DATA_BLOCK "DOOR_CLEANER_MOTOR_DB"	// DB 10
AUTHOR : Kamillas
VERSION : 0.1
  STRUCT
   DC_MTR_RDY_FOR_STA : BOOL ;	//DOOR CLEANER READY FOR START
   DC_MTR_UP_RUN_FB : BOOL ;	//DOOR CLEANER UP RUNNING FEED BACK
   DC_MTR_OLR_TRIP : BOOL ;	//DOOR CLEANER OVER LOAD TRIP
   DC_MTR_DN_RUN_FB : BOOL ;	//DOOR CLEANER DOWN RUNNING FEED BACK
   DC_MTR_AUTO_SS : BOOL ;	//DOOR CLEANER AUTO SELECTOR SWITCH
   DC_MTR_MAN_SS : BOOL ;	//DOOR CLEANER MANUAL SELECTOR SWITCH
   DC_MTR_UP_STA_PB : BOOL ;	//DOOR CLEANER UP START PUSH BUTTON
   DC_MTR_DN_STA_PB : BOOL ;	//DOOR CLEANER DOWN START PUSH BUTTON
   DC_MTR_STP_PB : BOOL ;	//DOOR CLEANER STOP PUSH BUTTON
   DC_MTR_HME_PB : BOOL ;	//DOOR CLEANER HOME PUSH BUTTON
   DC_MTR_UP_LS : BOOL ;	//DOOR CLEANER UP LIMIT SWITCH
   DC_MTR_DN_LS : BOOL ;	//DOOR CLEANER DOWN LIMIT SWITCH
   DC_MTR_HME_LS : BOOL ;	//DOOR CLEANER HOME LIMIT SWITCH
   CLN_OVN_DR_STA_PB : BOOL ;	//CLEAN OVEN DOOR START PUSH BUTTON
   CLN_OVN_DR_STP_PB : BOOL ;	//CLEAN OVEN DOOR STOP PUSH BUTTON
   DC_MTR_UP_ON_CMD : BOOL ;	//DOOR CLEANER UP ON COMMAND
   DC_MTR_DN_ON_CMD : BOOL ;	//DOOR CLEANER DOWN ON COMMAND
   DC_MTR_UP_IND : BOOL ;	//DOOR CLEANER UP INDICATOR
   DC_MTR_DN_IND : BOOL ;	//DOOR CLEANER DOWN INDICATOR
   DC_MTR_HME_IND : BOOL ;	//DOOR CLEANER HOME INDICATOR
   CLN_OVN_DR_AUTO_IND : BOOL ;	//CLEAN OVEN DOOR AUTO INDICATOR
   DC_MTR_FLT : BOOL ;	//DOOR COMPRESSOR MOTOR FAULT
   DC_MTR_FLT_TMR : INT ;	//DOOR COMPRESSOR MOTOR FAULT TIMER
   DC_MTR_FLT_GEN_TIME : INT  := 3;	//DOOR COMPRESSOR MOTOR FAULT GEMERATION TIME
   PULSE_1 : BOOL ;	//PULSE 1
   PULSE_2 : BOOL ;	//PULSE 2
   PULSE_3 : BOOL ;	//PULSE 3
   PULSE_4 : BOOL ;	//PULSE 4
   PULSE_5 : BOOL ;	//PULSE 5
   PULSE_6 : BOOL ;	//PULSE 6
   PULSE_7 : BOOL ;	//PULSE 7
   PULSE_8 : BOOL ;	//PULSE 8
   DC_MTR_ILK_BIT : BOOL ;	//DOOR CLEANER MOTOR INTERLOCK BIT
   DC_MTR_AUTO_STA_BIT : BOOL ;	//DOOR CLEANER MOTOR AUTO START BIT
   DC_MTR_HME_POS_BIT : BOOL ;	//DOOR CLEANER MOTOR HOME POSITION BIT
   DC_MTR_UP_DN_CNT_OVR : BOOL ;	//DOOR CLEANER MOTOR UP DOWN COUNT OVER
   DC_MTR_UP_DN_CNT : INT ;	//DOOR CLEANER UP DOWN COUNT
   DC_MTR_UP_DN_CNT_SET : INT  := 2;	//DOOR CLEANER MOTOR UP DOWN COUNT SET POINT
   DC_MTR_LOC_SS : BOOL ;	//DOOR CLEANER MOTOR LOCAL SELECTOR SWITCH
   DC_MTR_HME_ON_CMD : BOOL ;	//DOOR CLEANER HOME ON COMMAND
   DC_MTR_CLN_OVN_DOOR_IND : BOOL ;	//DOOR CLEANER - CLEAN OVEN DOOR INDICATOR
   TRA_SLOW_FWD_OP_CUT : BOOL ;	//TRAVEL SLOW FORWARD OUTPUT CUT
   TRA_SLOW_FWD_FLT_TMR : INT ;	//TRAVEL SLOW FORWARD FAULT TIMER
   TRA_SLOW_FWD_FLT_GEN : INT  := 8;	//TRAVEL SLOW FORWARD FAULT GENERATION TIME
   TRA_SLOW_FWD_OP_CT_TM : INT ;	//TRAVEL SLOW FORWARD OUTPUT CUT TIMER
   TRA_SLOW_FWD_FLT : BOOL ;	//TRAVEL SLOW FORWARD FAULT
   TRA_SLOW_AUTO_FWD_OVR : BOOL ;	//TRAVEL SLOW AUTO FORWARD OVER
   TRA_SLOW_AUTO_FWD_DEL : INT  := 3;	//TRAVEL SLOW AUTO FORWARD OVER DELAY
   TRA_SLOW_ATO_FWD_DL_T : INT ;	//TRAVEL SLOW AUTO FORWARD OVER DELAY TIMER
   TRA_SLOW_RET_OP_CUT : BOOL ;	//TRAVEL SLOW RETRACT OUTPUT CUT
   TRA_SLOW_RET_FLT_TMR : INT ;	//TRAVEL SLOW RETRACT FAULT TIMER
   TRA_SLOW_RET_FLT_GEN : INT  := 8;	//TRAVEL SLOW RETRACT FAULT GENERATION TIME
   TRA_SLOW_RET_OP_CT_TM : INT ;	//TRAVEL SLOW RETRACT OUTPUT CUT TIMER
   TRA_SLOW_RET_FLT : BOOL ;	//TRAVEL SLOW RETRACT FAULT
   TRA_SLOW_AUTO_RET_OVR : BOOL ;	//TRAVEL SLOW AUTO RETRACT OVER
   TRA_SLOW_AUTO_RET_DEL : INT  := 3;	//TRAVEL SLOW AUTO RETRACT OVER DELAY
   TRA_SLOW_ATO_RET_DL_T : INT ;	//TRAVEL SLOW AUTO RETRACT OVER DELAY TIMER
   TRA_NOR_FWD_OP_CUT : BOOL ;	//TRAVEL NORMAL FORWARD OUTPUT CUT
   TRA_NOR_FWD_FLT_TMR : INT ;	//TRAVEL NORMAL FORWARD FAULT TIMER
   TRA_NOR_FWD_FLT_GEN : INT  := 8;	//TRAVEL NORMAL FORWARD FAULT GENERATION TIME
   TRA_NOR_FWD_OP_CT_TM : INT ;	//TRAVEL NORMAL FORWARD OUTPUT CUT TIMER
   TRA_NOR_FWD_FLT : BOOL ;	//TRAVEL NORMAL FORWARD FAULT
   TRA_NOR_AUTO_FWD_OVR : BOOL ;	//TRAVEL NORMAL AUTO FORWARD OVER
   TRA_NOR_AUTO_FWD_DEL : INT  := 3;	//TRAVEL NORMAL AUTO FORWARD OVER DELAY
   TRA_NOR_ATO_FWD_DL_T : INT ;	//TRAVEL NORMAL AUTO FORWARD OVER DELAY TIMER
   TRA_NOR_RET_OP_CUT : BOOL ;	//TRAVEL NORMAL RETRACT OUTPUT CUT
   TRA_NOR_RET_FLT_TMR : INT ;	//TRAVEL NORMAL RETRACT FAULT TIMER
   TRA_NOR_RET_FLT_GEN : INT  := 8;	//TRAVEL NORMAL RETRACT FAULT GENERATION TIME
   TRA_NOR_RET_OP_CT_TM : INT ;	//TRAVEL NORMAL RETRACT OUTPUT CUT TIMER
   TRA_NOR_RET_FLT : BOOL ;	//TRAVEL NORMAL RETRACT FAULT
   TRA_NOR_AUTO_RET_OVR : BOOL ;	//TRAVEL NORMAL AUTO RETRACT OVER
   TRA_NOR_AUTO_RET_DEL : INT  := 3;	//TRAVEL NORMAL AUTO RETRACT OVER DELAY
   TRA_NOR_ATO_RET_DL_T : INT ;	//TRAVEL NORMAL AUTO RETRACT OVER DELAY TIMER
   TRA_SLOW_FWD_CMD : BOOL ;	//TRAVEL SLOW FORWARD COMMAND
   TRA_SLOW_RET_CMD : BOOL ;	//TRAVEL SLOW RETRACT COMMAND
   TRA_NOR_FWD_CMD : BOOL ;	//TRAVEL NORMAL FORWARD COMMAND
   TRA_NOR_RET_CMD : BOOL ;	//TRAVEL NORMAL RETRACT COMMAND
   TRA_RELIVE_CMD : BOOL ;	//TRAVEL RELIVE COOMMAND
   TRA_AUTO_FWD_CLN_POS_SET : BOOL ;	//TRAVEL AUTO FORWARD TO CLEANING POSITION SET
   TRA_AUTO_RET_SET : BOOL ;	//TRAVEL AUTO RETRACT SET
   TRA_CLN_POS_LS : BOOL ;	//TRAVEL CLEANING POSTION LIMIT SWITCH
   PULSE_9 : BOOL ;	//PULSE 9
   PULSE_10 : BOOL ;	//PULSE 10
   PULSE_11 : BOOL ;	//PULSE 11
   PULSE_12 : BOOL ;	//PULSE 12
   PULSE_13 : BOOL ;	//PULSE 13
   PULSE_14 : BOOL ;	//PULSE 14
   PULSE_15 : BOOL ;	//PULSE 15
   PULSE_16 : BOOL ;	//PULSE 16
   DC_MTR_HME_SET : BOOL ;	//TRAVEL AUTO HOME SET
   DC_MTR_AUTO_OPER_FIN : BOOL ;	//DOOR CLEANER MOTOR AUTO OPERATIONS FINISHED
   DC_AUTO_STOPPED : BOOL ;	//DOOR CLEANER OPERATIONS STOPED WHILE IN AUTO OPERATION
   DC_MTR_UP_LS_HOLD : BOOL ;	//UP LIMIT SWITCH HOLDING
   DC_MTR_DN_LS_HOLD : BOOL ;	//DOWN LIMIT SWITCH HOLDING
   DC_MTR_HME_LS_HOLD : BOOL ;	//HOME LIMIT SWITCH HOLDING
  END_STRUCT ;	
BEGIN
   DC_MTR_FLT_GEN_TIME := 3;
   DC_MTR_UP_DN_CNT_SET := 2;
   TRA_SLOW_FWD_FLT_GEN := 8;
   TRA_SLOW_AUTO_FWD_DEL := 3;
   TRA_SLOW_RET_FLT_GEN := 8;
   TRA_SLOW_AUTO_RET_DEL := 3;
   TRA_NOR_FWD_FLT_GEN := 8;
   TRA_NOR_AUTO_FWD_DEL := 3;
   TRA_NOR_RET_FLT_GEN := 8;
   TRA_NOR_AUTO_RET_DEL := 3;
END_DATA_BLOCK

DATA_BLOCK "WIN_CC_DB"	// DB 11
AUTHOR : Kamilas
VERSION : 0.1
  STRUCT
   MAIN_PWR_ON_PB : BOOL ;	//MAIN POWER ON PUSH BUTTON
   MAIN_PWR_OFF_PB : BOOL ;	//MAIN POWER OFF PUSH BUTTON
   MP_LAMP_TEST_PB : BOOL ;	//MAIN POWER LAMP TEST PUSH BUTTON
   MP_ALARM_ACK_PB : BOOL ;	//MAIN POWER ALARM ACKNOWLEDGE PUSH BUTTON
   CTRL_SELECTION_CD : BOOL ;	//CONTROL SELECTRION CD
   ALL_MECH_QUICK_STP : BOOL ;	//ALL MECHANICAL QUICK STOP
   REP_MAN_SS : BOOL ;	//REPAIR MANUAL SELECTION
   SEMI_AUTO_SS : BOOL ;	//SEMI AUTO SELECTION
   PUMP_1_RDY_FOR_STA : BOOL ;	//PUMP 1 READY FOR START
   PUMP_2_RDY_FOR_STA : BOOL ;	//PUMP 2 READY FOR START
   CIR_PUMP_RDY_FOR_STA : BOOL ;	//CIRCULATION PUMP READY FOR START
   COLR_FAN_RDY_FOR_STA : BOOL ;	//COOLER FAN READY FOR START
   CD_LCS_SS : BOOL ;	//CONTROL DESK / LOCAL CONTROL SELECTOR SWITCH
   HY_PUMP_1_2_SS : BOOL ;	//PUMP 1 OR 2 SELECTOR SWITCH
   HY_PUMP_1_STA_PB : BOOL ;	//PUMP 1 START PUSH BUTTON
   HY_PUMP_1_STP_PB : BOOL ;	//PUMP 1 STOP PUSH BUTTON
   HY_PUMP_2_STA_PB : BOOL ;	//PUMP 2 START PUSH BUTTON
   HY_PUMP_2_STP_PB : BOOL ;	//PUMP 2 STOP PUSH BUTTON
   HY_PUMP_1_2_SS_LCS : BOOL ;	//PUMP 1 OR 2 SELECTOR SWITCH LCS
   HY_PUMP_1_STA_PB_LCS : BOOL ;	//PUMP 1 START PUSH BUTTON LCS
   HY_PUMP_1_STP_PB_LCS : BOOL ;	//PUMP 1 STOP PUSH BUTTON LCS
   HY_PUMP_2_STA_PB_LCS : BOOL ;	//PUMP 2 START PUSH BUTTON LCS
   HY_PUMP_2_STP_PB_LCS : BOOL ;	//PUMP 2 STOP PUSH BUTTON LCS
   HY_CIR_PUMP_STA_PB_LCS : BOOL ;	//CIRCULATION PUMP START PUSH BUTTON LCS
   HY_CIR_PUMP_STP_PB_LCS : BOOL ;	//CIRCULATION PUMP STOP PUSH BUTTON LCS
   HY_COLR_FAN_STA_PB_LCS : BOOL ;	//COOLER FAN START PUSH BUTTON LCS
   HY_COLR_FAN_STP_PB_LCS : BOOL ;	//COOLER FAN STOP PUSH BUTTON LCS
   TRA_DRV_1_BRK_RDY_FOR_ST : BOOL ;	//TRAVEL GROUP 1 BREAK READY FOR START
   TRA_DRV_2_BRK_RDY_FOR_ST : BOOL ;	//TRAVEL GROUP 2 BREAK READY FOR START
   TRA_MODE_AUTO_MAN_SS : BOOL ;	//TRAVEL MODE AUTO/MANUAL BUTTON
   TRA_DRV_1_PROF_HARD_SS : BOOL ;	//TRAVEL DRIVE 1 PROFIBUS/HARD WIRE SELECTRO SWITCH
   TRA_DRV_1_RDY_FOR_STA : BOOL ;	//TRAVEL DRIVE 1 READY FOR START
   TRA_DRV_2_PROF_HARD_SS : BOOL ;	//TRAVEL DRIVE 2 PROFIBUS/HARD WIRE SELECTRO SWITCH
   TRA_DRV_2_RDY_FOR_STA : BOOL ;	//TRAVEL DRIVE 2 READY FOR START
   AC_MTR_RDY_FOR_STA : BOOL ;	//AIR COMPRESSOR MOTOR READY FOR START
   AC_MTR_STA_PB : BOOL ;	//AIR COMPRESSOR MOTOR START PUSH BUTTON
   AC_MTR_STP_PB : BOOL ;	//AIR COMPRESSOR MOTOR STOP PUSH BUTTON
   IDF_DRV_RDY_FOR_STA : BOOL ;	//ID FAN DRIVE READY FOR START
   WTR_PMP_MTR_RDY_FOR_STA : BOOL ;	//WATER PUMP MOTOR READY FOR START
   HOOD_STA_PB : BOOL ;	//HOOD START PUSH BUTTON
   HOOD_STP_PB : BOOL ;	//HOOD STOP PUSH BUTTON
   IDF_DRV_LS_HS_SEL : BOOL ;	//ID FAN DRIVE LOW SPEED/HIGH SPEED SELECTION
   DE_DOOR_EXT_LOC_SS : BOOL ;	//DOOR EXTRACTOR LOCAL SELECTOR SWITCH
   DE_DOOR_EXT_MAN_SS : BOOL ;	//DOOR EXTRACTOR MANUAL SELECTOR SWITCH
   DE_DOOR_EXT_AUTO_SS : BOOL ;	//DOOR EXTRACTOR AUTO SELECTOR SWITCH
   DE_DOOR_EXT_STP_PB : BOOL ;	//DOOR EXTRACTOR STOP PUSH BUTTON
   DE_SLEW_FWD_STA_PB : BOOL ;	//SLEW FORWARD START PUSH BUTTON
   DE_SLEW_RET_STA_PB : BOOL ;	//SLEW RETRACT START
   DE_VER_COMP_FWD_STA_PB : BOOL ;	//VERTICAL COMPENSATION FORWARD START PUSH BUTTON
   DE_VER_COMP_RET_STA_PB : BOOL ;	//VERTICAL COMPENSATION RETRACT START PUSH BUTTON
   DE_TRA_FWD_STA_PB : BOOL ;	//TRAVEL FORWARD START PUSH BUTTON
   DE_TRA_RET_STA_PB : BOOL ;	//TRAVEL RETRACT START PUSH BUTTON
   MAIN_STK_UP_STA_PB : BOOL ;	//MAIN STROKE UP START PUSH BUTTON
   MAIN_STK_DN_PB : BOOL ;	//MAIN STROKE DOWN START PUSH BUTTON
   FIN_STK_UP_STA_PB : BOOL ;	//FINAL STROKE UP START PUSH BUTTON
   FIN_STK_DN_PB : BOOL ;	//FINAL STROKE DOWN START PUSH BUTTON
   PRE_STK_UP_STA_PB : BOOL ;	//PRE STROKE UP START PUSH BUTTON
   PRE_STK_UP_DN_PB : BOOL ;	//PRE STROKE DOWN START PUSH BUTTON
   DR_SPNG_LK_STA_PB : BOOL ;	//DOOR SPRING PRESSURE START PUSH BUTTON
   DR_SPNG_UNLK_STA_PB : BOOL ;	//DOOR SPRING PRESSURE RELEASE START PUSH BUTTON
   DR_LCH_TURN_UP_PB : BOOL ;	//DOOR LATCH TURNING LOCK PUSH BUTTON
   DR_LCH_TURN_DN_PB : BOOL ;	//DOOR LATCH TURNING UNLOCK PUSH BUTTON
   JC_CRA_TRA_FWD_STA_PB : BOOL ;	//JAMB CLEANER CARRIAGE TRAVEL FORWARD PUSH BUTTON
   JC_CRA_TRA_RET_STA_PB : BOOL ;	//JAMB CLEANER CARRIAGE TRAVEL RETRACT PUSH BUTTON
   JC_VC_UP_STA_PB : BOOL ;	//JAMB CLEANER VERTICAL CLEANER UP START PUSH BUTTON
   JC_VC_DN_STA_PB : BOOL ;	//JAMB CLEANER VERTICAL CLEANER DOWN START PUSH BUTTON
   JC_STP_PB : BOOL ;	//JAMB CLEANER OPERATIONS STOP PUSH BUTTON
   JC_VC_HME_STA_PB : BOOL ;	//JAMB CLEANER VERTICAL CLEANER HOME START PUSH BUTTON
   CLN_OVN_JMB_STA_PB : BOOL ;	//CLEAN OVEN JAMB AUTO START PUSH BUTTON
   CLN_OVN_JMB_STP_PB : BOOL ;	//CLEAN OVEN JAMB AUTO STOP PUSH BUTTON
   JC_AUTO_SS : BOOL ;	//JAMB CLEANER AUTO MODE SELECTOR SWITCH
   JC_MAN_SS : BOOL ;	//JAMB CLEANER MANUAL MODE SELECTOR SWITCH
   JC_LOC_SS : BOOL ;	//JAMB CLEANER LOCAL MODE SELECTOR SWITCH
   JC_AUTO_STA_PB : BOOL ;	//JAMB CLEANER AUTO START PUSH BUTTON
   GC_AUTO_SS : BOOL ;	//GUIDE CAGE AUTO SELECTOR SWITCH
   GC_MAN_SS : BOOL ;	//GUIDE CAGE MANUAL SELECTOR SWITCH
   GC_TRA_FWD_STA_PB : BOOL ;	//GUIDE CAGE TRAVEL FORWARD START PUSH BUTTON
   GC_TRA_RET_STA_PB : BOOL ;	//GUIDE CAGE TRAVEL RETRACT START PUSH BUTTON
   GC_STP_PB : BOOL ;	//GUIDE CAGE AUTO STOP PUSH BUTTON
   GC_TRA_AUTO_STA_PB : BOOL ;	//GUIDE CAGE TRAVEL AUTO START PUSH BUTTON
   GC_TRA_AUTO_STP_PB : BOOL ;	//GUIDE CAGE TRAVEL AUTO STOP PUSH BUTTON
   GC_AUTO_STA_PB : BOOL ;	//GUIDE CAGE AUTO START PUSH BUTTON
   DC_MTR_RDY_FOR_STA : BOOL ;	//DOOR CLEANER READY FOR START
   DC_MTR_AUTO_SS : BOOL ;	//DOOR CLEANER AUTO SELECTOR SWITCH
   DC_MTR_MAN_SS : BOOL ;	//DOOR CLEANER MANUAL SELECTOR SWITCH
   DC_MTR_UP_STA_PB : BOOL ;	//DOOR CLEANER UP START PUSH BUTTON
   DC_MTR_DN_STA_PB : BOOL ;	//DOOR CLEANER DOWN START PUSH BUTTON
   DC_MTR_STP_PB : BOOL ;	//DOOR CLEANER STOP PUSH BUTTON
   DC_MTR_HME_PB : BOOL ;	//DOOR CLEANER HOME PUSH BUTTON
   CLN_OVN_DR_STA_PB : BOOL ;	//CLEAN OVEN DOOR START PUSH BUTTON
   CLN_OVN_DR_STP_PB : BOOL ;	//CLEAN OVEN DOOR STOP PUSH BUTTON
   DC_MTR_LOC_SS : BOOL ;	//DOOR CLEANER MOTOR LOCAL SELECTOR SWITCH
   SP_STP_PB : BOOL ;	//SERVICE PLATFORM STOP PUSH BUTTON
   SP_STA_PB : BOOL ;	//SERVICE PLATFORM START PUSH BUTTON
   EMG_ACCM_STA_PB_LCS : BOOL ;	//EMERGENCY ACCUMULATOR START PUSH BUTTON LCS
   EMG_ACCM_STP_PB_LCS : BOOL ;	//EMERGENCY ACCUMULATOR STOP PUSH BUTTON LCS
   EXT_OVN_DOR_STA_PB : BOOL ;	//EXTRACT OVEN DOOR START PUSH BUTTON
   EXT_RPL_FUNC_STP_PB : BOOL ;	//EXTRACT AND REPLACE FUNCTIONAL STOP PUSH BUTTON
   RPL_OVN_DOR_STA_PB : BOOL ;	//REPLACE OVEN DOOR START PUSH BUTTON
   ALL_OPER_IN_OPER_MODE : BOOL ;	//ALL OPERATION IN OPERATION MODE
   ALL_OPER_IN_REP_MODE : BOOL ;	//ALL OPERATION IN REPAIR MODE
   SP_TRA_FWD_STA_PB : BOOL ;	//SERVICE PLATFORM TRAVEL FORWARD START PUSH BUTTON
   SP_TRA_REV_STA_PB : BOOL ;	//SERVICE PLATFORM TRAVEL REVERSE START PUSH BUTTON
   EMERGENCY_STOP : BOOL ;	//EMERGENCY STOP
   HY_LAMP_TEST : BOOL ;	//HYDRALIC SYSTEM LAMP PUSH BUTTON
   SP_AUTO_STP_PB : BOOL ;	//SERVICE PLATFORM AUTO STOP PUSH BUTTON
   SP_TRA_AUTO_STA_PB : BOOL ;	//SERVICE PLATFORM TRAVEL AUTO START PUSH BUTTON
   SP_TRA_AUTO_STP_PB : BOOL ;	//SERVICE PLATFORM TRAVEL AUTO STOP PUSH BUTTON
   SP_AUTO_STA_PB : BOOL ;	//SERVICE PLATFORM AUTO START PUSH BUTTON
   SP_AUTO_SS : BOOL ;	//SERVICE PLATFORM AUTO MODE SELECTOR SWITCH
   SP_MAN_SS : BOOL ;	//SERVICE PLATFORM MANUAL MODE SELECTOR SWITCH
   MAIN_PWR_RDY_FOR_ON : BOOL ;	//MAIN POWER READY FOR ON
   MAIN_PWR_ON_FB : BOOL ;	//MAIN POWER ON FEED BACK
   CTRL_PWR_ON_FB : BOOL ;	//CONTROL POWER ON FEEDBACK
   PUMP_1_RUN_FB : BOOL ;	//PUMP 1 RUNNING FEEDBACK
   PUMP_1_OVR_LD_TRIP : BOOL ;	//PUMP 1 OVER LOAD TRIPPED
   PUMP_2_RUN_FB : BOOL ;	//PUMP 2 RUNNING FEEDBACK
   PUMP_2_OVR_LD_TRIP : BOOL ;	//PUMP 2 OVER LOAD TRIPPED
   CIR_PUMP_RUN_FB : BOOL ;	//CIRCULATION PUMP RUNNING FEEDBACK
   CIR_PUMP_OVR_LD_TRIP : BOOL ;	//CIRCULATION PUMP OVER LOAD TRIPPED
   COLR_FAN_RUN_FB : BOOL ;	//COOLER FAN RUNNING FEEDBACK
   COLR_FAN_OVR_LD_TRIP : BOOL ;	//COOLER FAN OVER LOAD TRIPPED
   SHT_OF_VLV_LIN_1_FUL_OPN : BOOL ;	//SHUT OFF VALVE IN LINE 1 - FULLY OPEN
   SHT_OF_VLV_LIN_2_FUL_OPN : BOOL ;	//SHUT OFF VALVE IN LINE 2 - FULLY OPEN
   LOW_OIL_TEMP : BOOL ;	//LOW OIL TEMPERATURE - THERMOSTAT
   HIGH_OIL_TEMP : BOOL ;	//HIGH OIL TEMPERATURE - THERMOSTAT
   MAX_OIL_TEMP : BOOL ;	//MAXIMUM OIL TEMPERATURE - THERMOSTAT
   LOW_OIL_LEVEL : BOOL ;	//LOW OIL LEVEL - FLOAT SWITCH
   MIN_OIL_LEVEL : BOOL ;	//MINIMUM OIL LEVEL - FLOAT SWITCH
   RET_LIN_FLTR_CKD : BOOL ;	//RETURN LINE FILTER CHOKED
   TRA_DRV_1_ON_FB : BOOL ;	//TRAVEL DRIVE 1 ON FEEDBACK
   TRA_DRV_1_TRP_FB : BOOL ;	//TRAVEL DRIVE 1 TRIP FEEDBACK
   SLEW_SLOW_FWD_LS : BOOL ;	//SLEW SLOW FORWARD LIMIT SWITCH
   SLEW_SLOW_RET_LS : BOOL ;	//SLEW SLOW RETRACT LIMIT SWITCH
   SLEW_NOR_FWD_LS : BOOL ;	//SLEW NORMAL FORWARD LIMIT SWITCH
   SLEW_NOR_RET_LS : BOOL ;	//SLEW NORMAL RETRACT LIMIT SWITCH
   TRA_SLOW_FWD_LS : BOOL ;	//TRAVEL SLOW FORWARD LIMIT  SWITCH
   TRA_SLOW_RET_LS : BOOL ;	//TRAVEL SLOW RETRACT LIMIT  SWITCH
   TRA_FWD_LS : BOOL ;	//TRAVEL FORWARD LIMIT SWIITCH
   TRA_RET_LS : BOOL ;	//TRAVEL RETRACT LIMIT SWIITCH
   FOR_LS_TRAVEL : BOOL ;	//FORWARD LIMIT SWITCH TRAVEL
   DOOR_ON_HOOK_LS : BOOL ;	//DOOR ON HOOK LIMITSWTCH
   JC_CAR_TRA_FWD_LS : BOOL ;	//JAMB CLEANER CARRIAGE TRAVEL FORWARD LIMIT SWITCH
   JC_CAR_TRA_RET_LS : BOOL ;	//JAMB CLEANER CARRIAGE TRAVEL RETRACT LIMIT SWITCH
   JC_VER_CLNR_UP_LS : BOOL ;	//JAMB CLEANER VERTICAL CLEANER UP LIMIT SWITCH
   JC_VER_CLNR_DN_LS : BOOL ;	//JAMB CLEANER VERTICAL CLEANER DOWN LIMIT SWITCH
   JC_VER_CLNR_HME_LS : BOOL ;	//JAMB CLEANER VERTICAL CLEANER HOME LIMIT SWITCH
   DC_MTR_UP_LS : BOOL ;	//DOOR CLEANER UP LIMIT SWITCH
   DC_MTR_DN_LS : BOOL ;	//DOOR CLEANER DOWN LIMIT SWITCH
   AC_MTR_RUN_FB : BOOL ;	//AIR COMPRESSOR MOTOR RUN FEED BACK
   AC_MTR_OLR_TRIP_FB : BOOL ;	//AIR COMPRESSOR MOTOR TRIP FEED BACK
   GC_TRA_FWD_LS : BOOL ;	//GUIDE CAGE TRAVEL FORWARD LIMIT SWITCH
   GC_TRA_RET_LS : BOOL ;	//GUIDE CAGE TRAVEL RETRACT LIMIT SWITCH
   TRA_JOY_STK_FWD_POS : BOOL ;	//TRAVEL JOY STICK FOWRWARD POSITION
   TRA_JOY_STK_REV_POS : BOOL ;	//TRAVEL JOY DEAD REVERSE POSITION
   TRA_JOY_STK_HME_POS : BOOL ;	//TRAVEL JOY STICK HOME POSITION
   TRA_JOY_STK_DED_MAN_BTN : BOOL ;	//TRAVEL JOY DEAD MAN BUTTON
   TRA_DRV_2_ON_FB : BOOL ;	//TRAVEL DRIVE 2 ON FEEDBACK
   TRA_DRV_2_TRP_FB : BOOL ;	//TRAVEL DRIVE 2 TRIP FEEDBACK
   DC_MTR_HME_LS : BOOL ;	//DOOR CLEANER HOME LIMIT SWITCH
   LAMP_TEST_PB : BOOL ;	//LAMP TEST PUSH BUTTON
   q : BOOL ;
   W : BOOL ;
   E : BOOL ;
   R : BOOL ;
   T : BOOL ;
   Y : BOOL ;
   U : BOOL ;
   REPR_OPER_MODE_SS : BOOL ;
   q1 : BOOL ;
   W1 : BOOL ;
   E1 : BOOL ;
   R1 : BOOL ;
   T1 : BOOL ;
   Y1 : BOOL ;
   U1 : BOOL ;
   TRAV_AUTO_MAN_SS : BOOL ;
   q11 : BOOL ;
   W11 : BOOL ;
   E11 : BOOL ;
   R11 : BOOL ;
   T11 : BOOL ;
   Y11 : BOOL ;
   U11 : BOOL ;
   SP_AUTO_MAN_SS : BOOL ;
   q111 : BOOL ;
   W111 : BOOL ;
   E111 : BOOL ;
   R111 : BOOL ;
   T111 : BOOL ;
   Y111 : BOOL ;
   U111 : BOOL ;
   GC_AUTO_MAN_SS : BOOL ;
   q1111 : BOOL ;
   W1111 : BOOL ;
   E1111 : BOOL ;
   R1111 : BOOL ;
   T1111 : BOOL ;
   Y1111 : BOOL ;
   U1111 : BOOL ;
   DC_AUTO_MAN_SS : BOOL ;
   q11111 : BOOL ;
   W11111 : BOOL ;
   E11111 : BOOL ;
   R11111 : BOOL ;
   T11111 : BOOL ;
   Y11111 : BOOL ;
   U11111 : BOOL ;
   JC_AUTO_MAN_SS : BOOL ;
   q111111 : BOOL ;
   W111111 : BOOL ;
   E111111 : BOOL ;
   R111111 : BOOL ;
   T111111 : BOOL ;
   Y111111 : BOOL ;
   U111111 : BOOL ;
   DE_AUTO_MAN_SS : BOOL ;
   q1111111 : BOOL ;
   W1111111 : BOOL ;
   E1111111 : BOOL ;
   R1111111 : BOOL ;
   T1111111 : BOOL ;
   Y1111111 : BOOL ;
   U1111111 : BOOL ;
   PUMP_CD_LCS_SS : BOOL ;
   q11111111 : BOOL ;
   W11111111 : BOOL ;
   E11111111 : BOOL ;
   R11111111 : BOOL ;
   T11111111 : BOOL ;
   Y11111111 : BOOL ;
   U11111111 : BOOL ;
   PUMP_1_2_SS : BOOL ;
   A : BOOL ;
   S : BOOL ;
   D : BOOL ;
   F : BOOL ;
   G : BOOL ;
   H : BOOL ;
   J : BOOL ;
   ID_FAN_HS_LS_SEL : BOOL ;
   A1 : BOOL ;
   S1 : BOOL ;
   D1 : BOOL ;
   F1 : BOOL ;
   G1 : BOOL ;
   H1 : BOOL ;
   J1 : BOOL ;
   JMB_CLN_HME_STA_PB : BOOL ;
  END_STRUCT ;	
BEGIN
END_DATA_BLOCK

DATA_BLOCK "CMD_FROM_TATA"	// DB 12
VERSION : 0.1
  STRUCT
   GC_OnBord_STATUS_BIT : STRUCT
    PUSH_PERM : BOOL ;	//Pushing interlock OK
    GC_LT_MODE : BOOL ;	//Long travel in auto or in man
    GC_TRAVEL_FWD : BOOL ;	//FWD over profibus
    GC_TRAVEL_REV : BOOL ;	//REV over profibus
    GC_TRAVEL_START : BOOL ;	//START over profibus
    GC_TRAVEL_STOP : BOOL ;	//STOP  over profibus
    SpareBit_1 : BOOL ;
    HOOD_SYS_ON_CMD : BOOL ;	//HOOD SYSTEM ON COMMAND
    GUIDE_CAGE_PERM : BOOL ;	//GUIDE CAGE PERMISSION
    SpareBit_4 : BOOL ;
    SpareBit_5 : BOOL ;
    SpareBit_6 : BOOL ;
    SpareBit_7 : BOOL ;
    SpareBit_8 : BOOL ;
    SpareBit_9 : BOOL ;
    SpareBit_10 : BOOL ;
    GC_SPEED_REF : INT ;	//Reserve for LT motion (spd_ref) over profibus
    SATA : ARRAY  [1 .. 7 ] OF INT ;
   END_STRUCT ;
  END_STRUCT ;	
BEGIN
END_DATA_BLOCK

DATA_BLOCK "FB_TO_TATA"	// DB 13
VERSION : 0.1
  STRUCT
   GC_MACHINE_STATUS_BIT : STRUCT
    COKE_SIDE_DOOR_CL : BOOL ;
    COKE_SIDE_DOOR_OP : BOOL ;
    GC_DRV_STATUS : BOOL ;
    GC_DRV_FWD : BOOL ;
    GC_DRV_REV : BOOL ;
    GC_PERM : BOOL ;
    GC_STATUS : BOOL ;
    SpareBit_2 : BOOL ;
    SpareBit_3 : BOOL ;
    SpareBit_4 : BOOL ;
    SpareBit_5 : BOOL ;
    SpareBit_6 : BOOL ;
    SpareBit_7 : BOOL ;
    SpareBit_8 : BOOL ;
    SpareBit_9 : BOOL ;
    SpareBit_10 : BOOL ;
    GC_SPEED : REAL ;
    Spare_Int0 : INT ;
    Spare_Int1 : INT ;
    SATA : ARRAY  [1 .. 4 ] OF INT ;
   END_STRUCT ;
  END_STRUCT ;	
BEGIN
END_DATA_BLOCK

DATA_BLOCK "TATA_COMMUNICATION_DB"	// DB 14
VERSION : 0.1
  STRUCT
   TATA_DATA_READ_ERROR : INT ;	//TATA PLC DATA READ ERROR
   TATA_DATA_WRITE_ERROR : INT ;	//TATA PLC DATA WRITE ERROR
   DR_OPN_LCH_TIMER : INT ;	//DOOR OPEN BIT LATCH TIMER
   DR_OPN_LCH_TIME : INT  := 5;	//DOOR OPEN BIT LATCH TIME
   DR_CLS_LCH_TIMER : INT ;	//DOOR CLOSE BIT LATCH TIMER
   DR_CLS_LCH_TIME : INT  := 5;	//DOOR CLOSE BIT LATCH TIME
   PUSLE_1 : BOOL ;	//PUSLE 1
   PUSLE_2 : BOOL ;	//PUSLE 2
   PUSLE_3 : BOOL ;	//PUSLE 3
   PUSLE_4 : BOOL ;	//PUSLE 4
   PUSLE_5 : BOOL ;	//PUSLE 5
   PUSLE_6 : BOOL ;	//PUSLE 6
   PUSLE_7 : BOOL ;	//PUSLE 7
   PUSLE_8 : BOOL ;	//PUSLE 8
  END_STRUCT ;	
BEGIN
   DR_OPN_LCH_TIME := 5;
   DR_CLS_LCH_TIME := 5;
END_DATA_BLOCK

ORGANIZATION_BLOCK "MAIN_PROGRAM"	// OB 1
AUTHOR : Kamillas
VERSION : 0.1
BEGIN
// (block stored without names or comments; labels and parameter names are numbered)
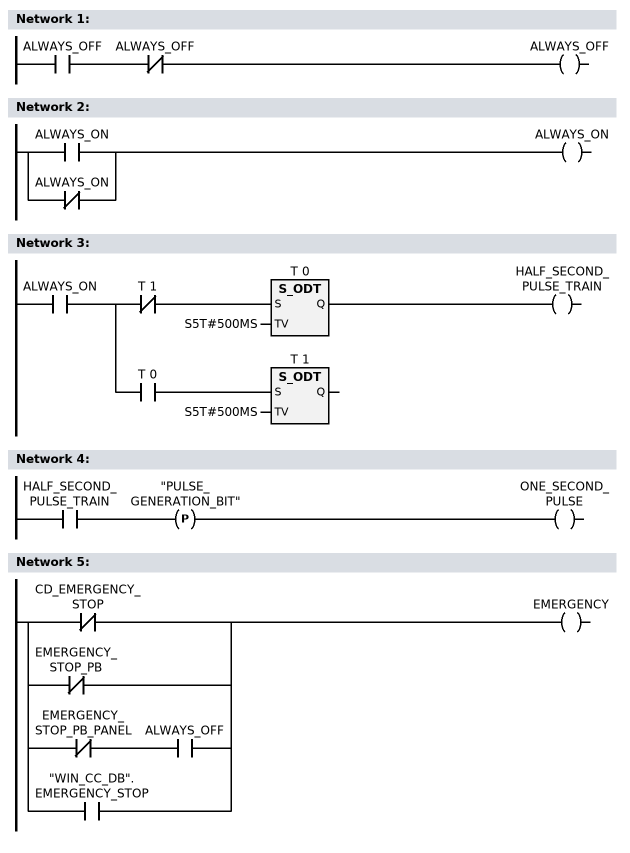
NETWORK
TITLE =
      A     "ALWAYS_OFF";
      AN    "ALWAYS_OFF";
      =     "ALWAYS_OFF";
NETWORK
TITLE =
      O     "ALWAYS_ON";
      ON    "ALWAYS_ON";
      =     "ALWAYS_ON";
NETWORK
TITLE =
      A     "ALWAYS_ON";
      =     L 20.0;
      A     L 20.0;
      AN    T 1;
      L     S5T#500MS;
      SD    T 0;
      NOP   0;
      NOP   0;
      NOP   0;
      A     T 0;
      =     "HALF_SECOND_PULSE_TRAIN";
      A     L 20.0;
      A     T 0;
      L     S5T#500MS;
      SD    T 1;
      NOP   0;
      NOP   0;
      NOP   0;
      NOP   0;
NETWORK
TITLE =
      A     "HALF_SECOND_PULSE_TRAIN";
      FP    "PULSE_GENERATION_BIT";
      =     "ONE_SECOND_PULSE";
NETWORK
TITLE =
      ON    "CD_EMERGENCY_STOP";
      ON    "EMERGENCY_STOP_PB";
      O;
      AN    "EMERGENCY_STOP_PB_PANEL";
      A     "ALWAYS_OFF";
      O     "WIN_CC_DB".EMERGENCY_STOP;
      =     "EMERGENCY";
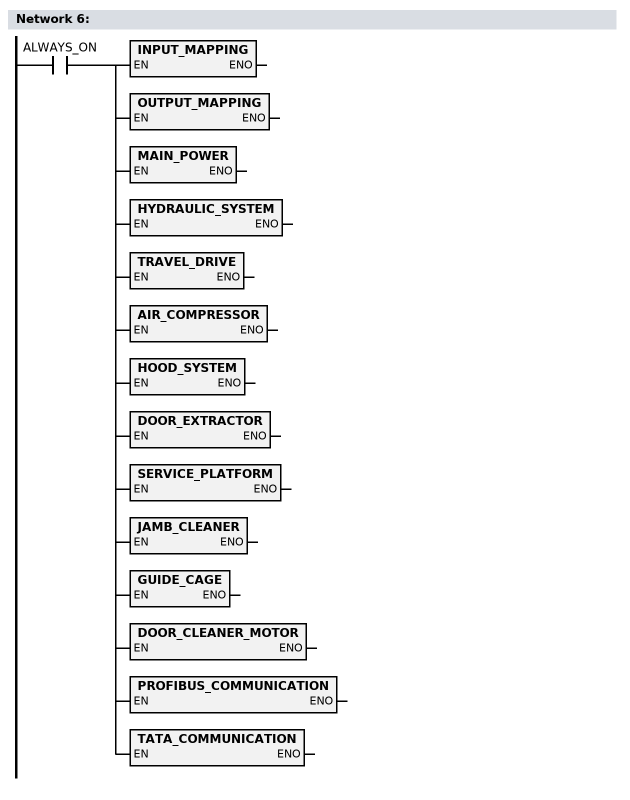
NETWORK
TITLE =
      A     "ALWAYS_ON";
      =     L 20.0;
      A     L 20.0;
      JNB   M001;
      CALL  "INPUT_MAPPING";
M001: NOP   0;
      A     L 20.0;
      JNB   M002;
      CALL  "OUTPUT_MAPPING";
M002: NOP   0;
      A     L 20.0;
      JNB   M003;
      CALL  "MAIN_POWER";
M003: NOP   0;
      A     L 20.0;
      JNB   M004;
      CALL  "HYDRAULIC_SYSTEM";
M004: NOP   0;
      A     L 20.0;
      JNB   M005;
      CALL  "TRAVEL_DRIVE";
M005: NOP   0;
      A     L 20.0;
      JNB   M006;
      CALL  "AIR_COMPRESSOR";
M006: NOP   0;
      A     L 20.0;
      JNB   M007;
      CALL  "HOOD_SYSTEM";
M007: NOP   0;
      A     L 20.0;
      JNB   M008;
      CALL  "DOOR_EXTRACTOR";
M008: NOP   0;
      A     L 20.0;
      JNB   M009;
      CALL  "SERVICE_PLATFORM";
M009: NOP   0;
      A     L 20.0;
      JNB   M010;
      CALL  "JAMB_CLEANER";
M010: NOP   0;
      A     L 20.0;
      JNB   M011;
      CALL  "GUIDE_CAGE";
M011: NOP   0;
      A     L 20.0;
      JNB   M012;
      CALL  "DOOR_CLEANER_MOTOR";
M012: NOP   0;
      A     L 20.0;
      JNB   M013;
      CALL  "PROFIBUS_COMMUNICATION";
M013: NOP   0;
      A     L 20.0;
      JNB   M014;
      CALL  "TATA_COMMUNICATION";
M014: NOP   0;
END_ORGANIZATION_BLOCK

ORGANIZATION_BLOCK "I/O_FLT1"	// OB 82
AUTHOR : Kamillas
VERSION : 0.1
BEGIN
// (block stored without names or comments; labels and parameter names are numbered)
END_ORGANIZATION_BLOCK

ORGANIZATION_BLOCK "RACK_FLT"	// OB 86
AUTHOR : Kamillas
VERSION : 0.1
BEGIN
// (block stored without names or comments; labels and parameter names are numbered)
END_ORGANIZATION_BLOCK

ORGANIZATION_BLOCK "PROG_ERR"	// OB 121
AUTHOR : Kamillas
VERSION : 0.1
BEGIN
// (block stored without names or comments; labels and parameter names are numbered)
END_ORGANIZATION_BLOCK

ORGANIZATION_BLOCK "MOD_ERR"	// OB 122
AUTHOR : Kamillas
VERSION : 0.1
BEGIN
// (block stored without names or comments; labels and parameter names are numbered)
END_ORGANIZATION_BLOCK

FUNCTION FC 1 : VOID
AUTHOR : Kamillas
VERSION : 0.1
BEGIN
// (block stored without names or comments; labels and parameter names are numbered)
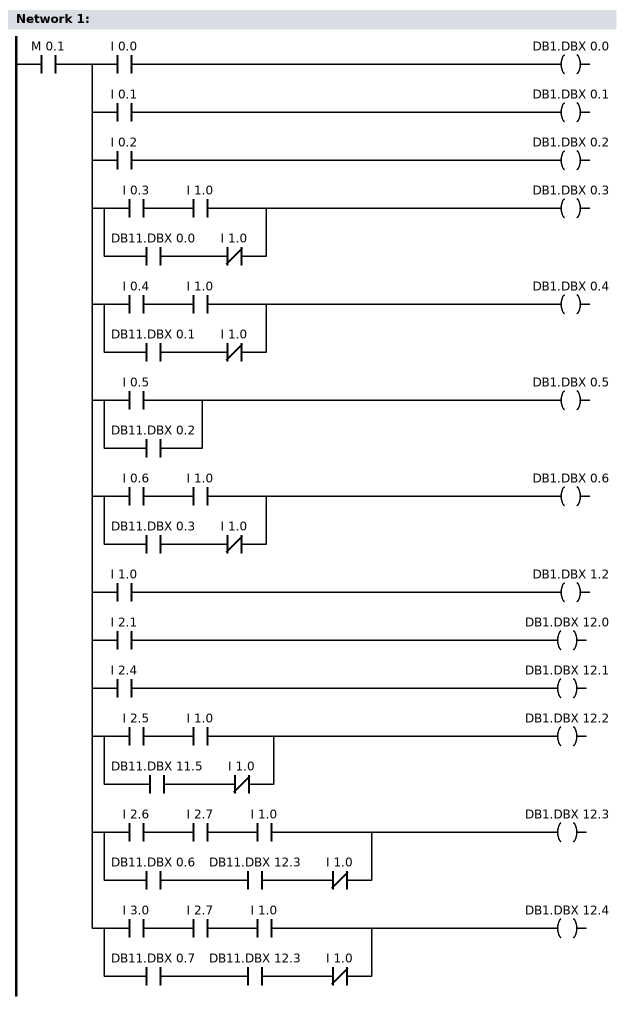
NETWORK
TITLE =
      A     M 0.1;
      =     L 0.0;
      A     L 0.0;
      A     I 0.0;
      =     DB1.DBX 0.0;
      A     L 0.0;
      A     I 0.1;
      =     DB1.DBX 0.1;
      A     L 0.0;
      A     I 0.2;
      =     DB1.DBX 0.2;
      A     L 0.0;
      A(;
      A     I 0.3;
      A     I 1.0;
      O;
      A     DB11.DBX 0.0;
      AN    I 1.0;
      );
      =     DB1.DBX 0.3;
      A     L 0.0;
      A(;
      A     I 0.4;
      A     I 1.0;
      O;
      A     DB11.DBX 0.1;
      AN    I 1.0;
      );
      =     DB1.DBX 0.4;
      A     L 0.0;
      A(;
      O     I 0.5;
      O     DB11.DBX 0.2;
      );
      =     DB1.DBX 0.5;
      A     L 0.0;
      A(;
      A     I 0.6;
      A     I 1.0;
      O;
      A     DB11.DBX 0.3;
      AN    I 1.0;
      );
      =     DB1.DBX 0.6;
      A     L 0.0;
      A     I 1.0;
      =     DB1.DBX 1.2;
      A     L 0.0;
      A     I 2.1;
      =     DB1.DBX 12.0;
      A     L 0.0;
      A     I 2.4;
      =     DB1.DBX 12.1;
      A     L 0.0;
      A(;
      A     I 2.5;
      A     I 1.0;
      O;
      A     DB11.DBX 11.5;
      AN    I 1.0;
      );
      =     DB1.DBX 12.2;
      A     L 0.0;
      A(;
      A     I 2.6;
      A     I 2.7;
      A     I 1.0;
      O;
      A     DB11.DBX 0.6;
      A     DB11.DBX 12.3;
      AN    I 1.0;
      );
      =     DB1.DBX 12.3;
      A     L 0.0;
      A(;
      A     I 3.0;
      A     I 2.7;
      A     I 1.0;
      O;
      A     DB11.DBX 0.7;
      A     DB11.DBX 12.3;
      AN    I 1.0;
      );
      =     DB1.DBX 12.4;
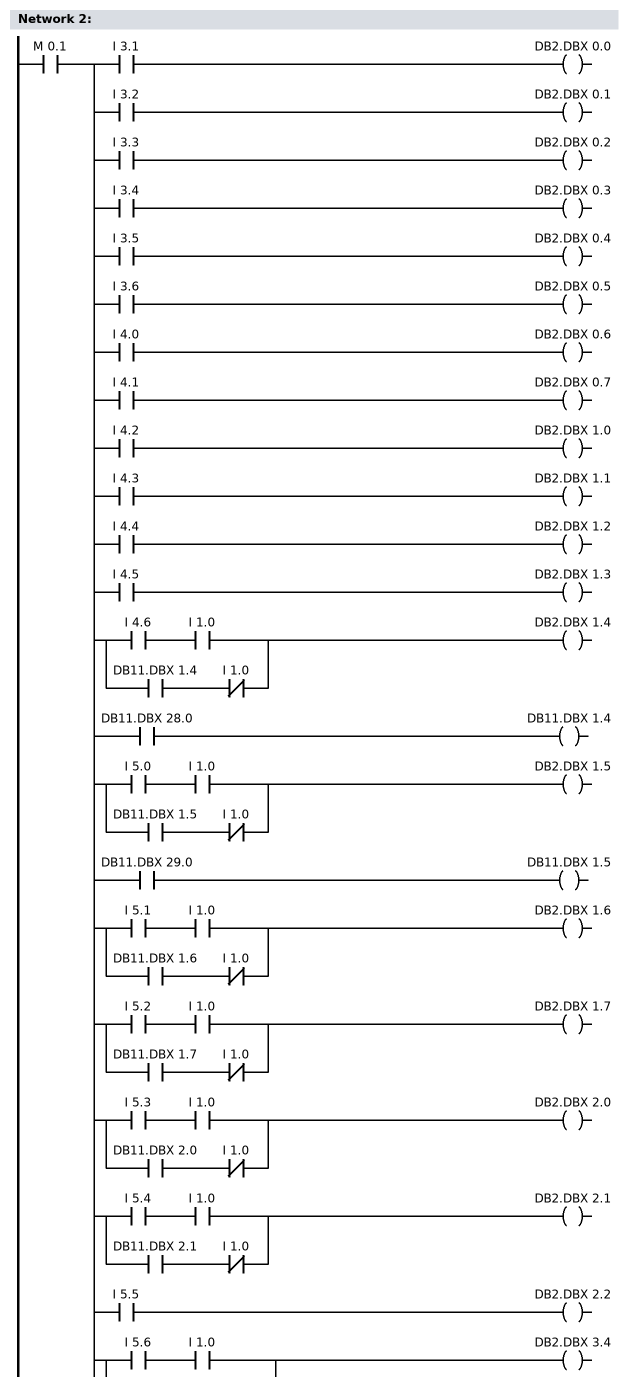
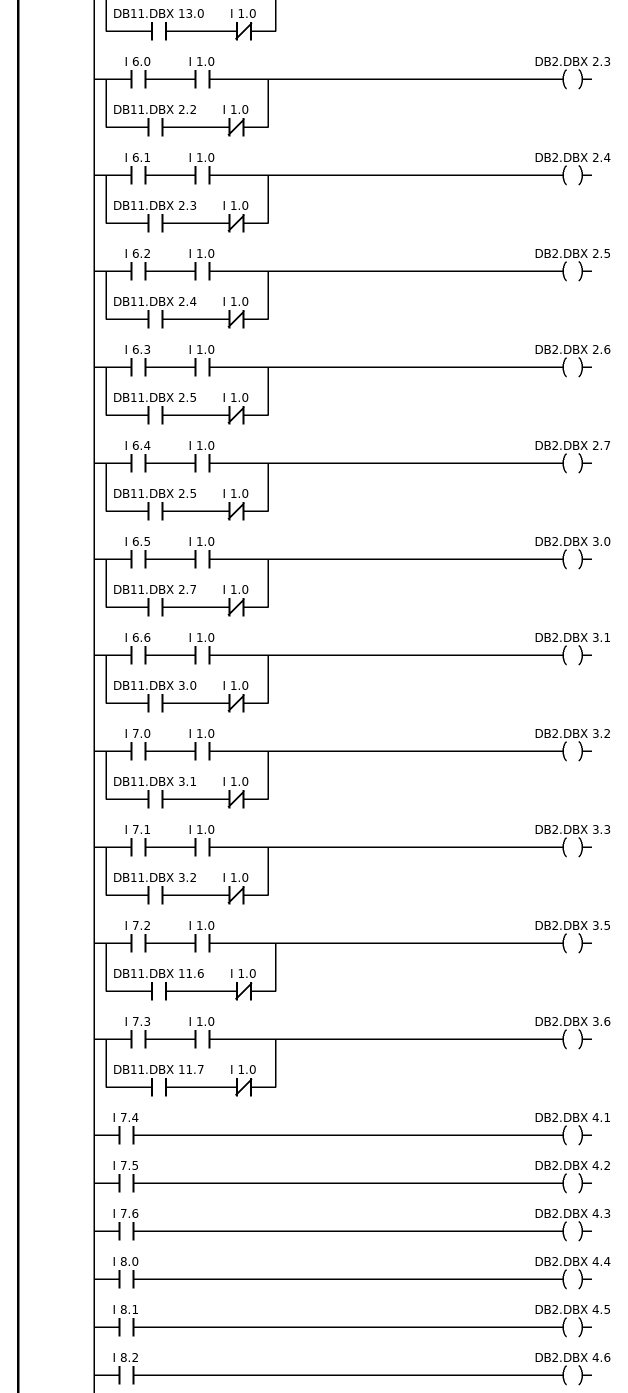
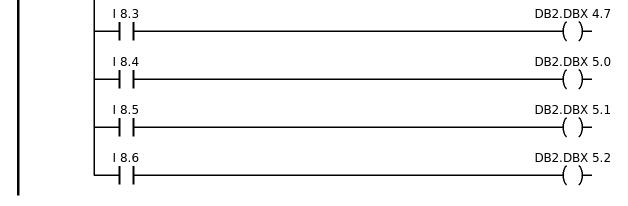
NETWORK
TITLE =
      A     M 0.1;
      =     L 0.0;
      A     L 0.0;
      A     I 3.1;
      =     DB2.DBX 0.0;
      A     L 0.0;
      A     I 3.2;
      =     DB2.DBX 0.1;
      A     L 0.0;
      A     I 3.3;
      =     DB2.DBX 0.2;
      A     L 0.0;
      A     I 3.4;
      =     DB2.DBX 0.3;
      A     L 0.0;
      A     I 3.5;
      =     DB2.DBX 0.4;
      A     L 0.0;
      A     I 3.6;
      =     DB2.DBX 0.5;
      A     L 0.0;
      A     I 4.0;
      =     DB2.DBX 0.6;
      A     L 0.0;
      A     I 4.1;
      =     DB2.DBX 0.7;
      A     L 0.0;
      A     I 4.2;
      =     DB2.DBX 1.0;
      A     L 0.0;
      A     I 4.3;
      =     DB2.DBX 1.1;
      A     L 0.0;
      A     I 4.4;
      =     DB2.DBX 1.2;
      A     L 0.0;
      A     I 4.5;
      =     DB2.DBX 1.3;
      A     L 0.0;
      A(;
      A     I 4.6;
      A     I 1.0;
      O;
      A     DB11.DBX 1.4;
      AN    I 1.0;
      );
      =     DB2.DBX 1.4;
      A     L 0.0;
      A     DB11.DBX 28.0;
      =     DB11.DBX 1.4;
      A     L 0.0;
      A(;
      A     I 5.0;
      A     I 1.0;
      O;
      A     DB11.DBX 1.5;
      AN    I 1.0;
      );
      =     DB2.DBX 1.5;
      A     L 0.0;
      A     DB11.DBX 29.0;
      =     DB11.DBX 1.5;
      A     L 0.0;
      A(;
      A     I 5.1;
      A     I 1.0;
      O;
      A     DB11.DBX 1.6;
      AN    I 1.0;
      );
      =     DB2.DBX 1.6;
      A     L 0.0;
      A(;
      A     I 5.2;
      A     I 1.0;
      O;
      A     DB11.DBX 1.7;
      AN    I 1.0;
      );
      =     DB2.DBX 1.7;
      A     L 0.0;
      A(;
      A     I 5.3;
      A     I 1.0;
      O;
      A     DB11.DBX 2.0;
      AN    I 1.0;
      );
      =     DB2.DBX 2.0;
      A     L 0.0;
      A(;
      A     I 5.4;
      A     I 1.0;
      O;
      A     DB11.DBX 2.1;
      AN    I 1.0;
      );
      =     DB2.DBX 2.1;
      A     L 0.0;
      A     I 5.5;
      =     DB2.DBX 2.2;
      A     L 0.0;
      A(;
      A     I 5.6;
      A     I 1.0;
      O;
      A     DB11.DBX 13.0;
      AN    I 1.0;
      );
      =     DB2.DBX 3.4;
      A     L 0.0;
      A(;
      A     I 6.0;
      A     I 1.0;
      O;
      A     DB11.DBX 2.2;
      AN    I 1.0;
      );
      =     DB2.DBX 2.3;
      A     L 0.0;
      A(;
      A     I 6.1;
      A     I 1.0;
      O;
      A     DB11.DBX 2.3;
      AN    I 1.0;
      );
      =     DB2.DBX 2.4;
      A     L 0.0;
      A(;
      A     I 6.2;
      A     I 1.0;
      O;
      A     DB11.DBX 2.4;
      AN    I 1.0;
      );
      =     DB2.DBX 2.5;
      A     L 0.0;
      A(;
      A     I 6.3;
      A     I 1.0;
      O;
      A     DB11.DBX 2.5;
      AN    I 1.0;
      );
      =     DB2.DBX 2.6;
      A     L 0.0;
      A(;
      A     I 6.4;
      A     I 1.0;
      O;
      A     DB11.DBX 2.5;
      AN    I 1.0;
      );
      =     DB2.DBX 2.7;
      A     L 0.0;
      A(;
      A     I 6.5;
      A     I 1.0;
      O;
      A     DB11.DBX 2.7;
      AN    I 1.0;
      );
      =     DB2.DBX 3.0;
      A     L 0.0;
      A(;
      A     I 6.6;
      A     I 1.0;
      O;
      A     DB11.DBX 3.0;
      AN    I 1.0;
      );
      =     DB2.DBX 3.1;
      A     L 0.0;
      A(;
      A     I 7.0;
      A     I 1.0;
      O;
      A     DB11.DBX 3.1;
      AN    I 1.0;
      );
      =     DB2.DBX 3.2;
      A     L 0.0;
      A(;
      A     I 7.1;
      A     I 1.0;
      O;
      A     DB11.DBX 3.2;
      AN    I 1.0;
      );
      =     DB2.DBX 3.3;
      A     L 0.0;
      A(;
      A     I 7.2;
      A     I 1.0;
      O;
      A     DB11.DBX 11.6;
      AN    I 1.0;
      );
      =     DB2.DBX 3.5;
      A     L 0.0;
      A(;
      A     I 7.3;
      A     I 1.0;
      O;
      A     DB11.DBX 11.7;
      AN    I 1.0;
      );
      =     DB2.DBX 3.6;
      A     L 0.0;
      A     I 7.4;
      =     DB2.DBX 4.1;
      A     L 0.0;
      A     I 7.5;
      =     DB2.DBX 4.2;
      A     L 0.0;
      A     I 7.6;
      =     DB2.DBX 4.3;
      A     L 0.0;
      A     I 8.0;
      =     DB2.DBX 4.4;
      A     L 0.0;
      A     I 8.1;
      =     DB2.DBX 4.5;
      A     L 0.0;
      A     I 8.2;
      =     DB2.DBX 4.6;
      A     L 0.0;
      A     I 8.3;
      =     DB2.DBX 4.7;
      A     L 0.0;
      A     I 8.4;
      =     DB2.DBX 5.0;
      A     L 0.0;
      A     I 8.5;
      =     DB2.DBX 5.1;
      A     L 0.0;
      A     I 8.6;
      =     DB2.DBX 5.2;
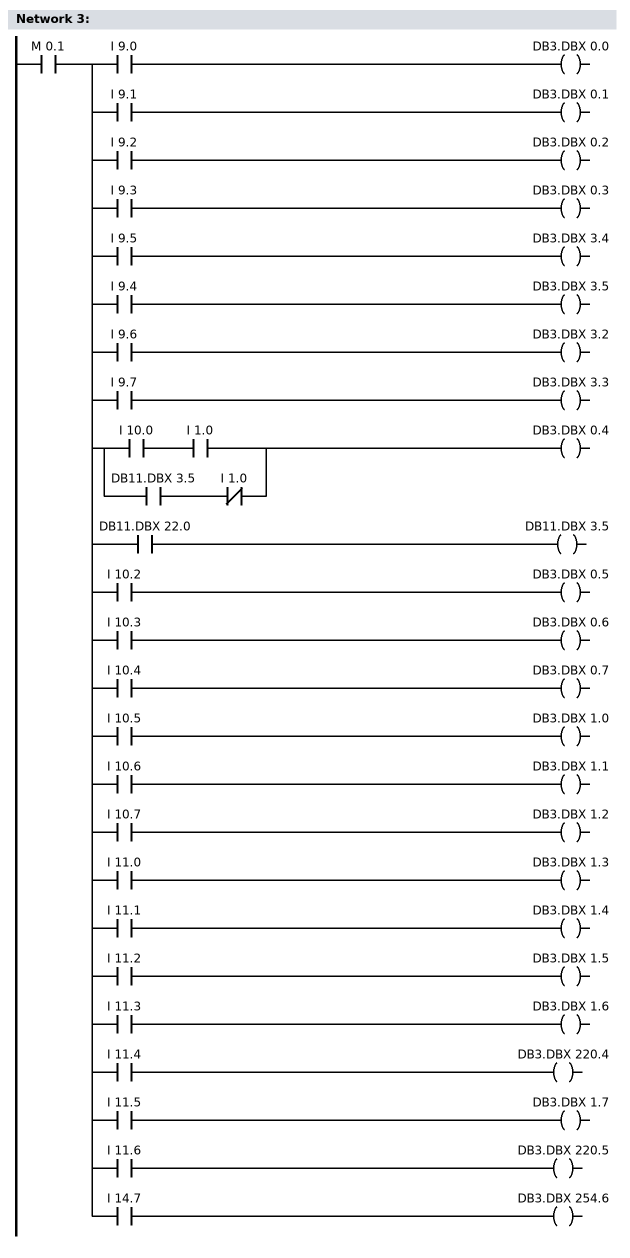
NETWORK
TITLE =
      A     M 0.1;
      =     L 0.0;
      A     L 0.0;
      A     I 9.0;
      =     DB3.DBX 0.0;
      A     L 0.0;
      A     I 9.1;
      =     DB3.DBX 0.1;
      A     L 0.0;
      A     I 9.2;
      =     DB3.DBX 0.2;
      A     L 0.0;
      A     I 9.3;
      =     DB3.DBX 0.3;
      A     L 0.0;
      A     I 9.5;
      =     DB3.DBX 3.4;
      A     L 0.0;
      A     I 9.4;
      =     DB3.DBX 3.5;
      A     L 0.0;
      A     I 9.6;
      =     DB3.DBX 3.2;
      A     L 0.0;
      A     I 9.7;
      =     DB3.DBX 3.3;
      A     L 0.0;
      A(;
      A     I 10.0;
      A     I 1.0;
      O;
      A     DB11.DBX 3.5;
      AN    I 1.0;
      );
      =     DB3.DBX 0.4;
      A     L 0.0;
      A     DB11.DBX 22.0;
      =     DB11.DBX 3.5;
      A     L 0.0;
      A     I 10.2;
      =     DB3.DBX 0.5;
      A     L 0.0;
      A     I 10.3;
      =     DB3.DBX 0.6;
      A     L 0.0;
      A     I 10.4;
      =     DB3.DBX 0.7;
      A     L 0.0;
      A     I 10.5;
      =     DB3.DBX 1.0;
      A     L 0.0;
      A     I 10.6;
      =     DB3.DBX 1.1;
      A     L 0.0;
      A     I 10.7;
      =     DB3.DBX 1.2;
      A     L 0.0;
      A     I 11.0;
      =     DB3.DBX 1.3;
      A     L 0.0;
      A     I 11.1;
      =     DB3.DBX 1.4;
      A     L 0.0;
      A     I 11.2;
      =     DB3.DBX 1.5;
      A     L 0.0;
      A     I 11.3;
      =     DB3.DBX 1.6;
      A     L 0.0;
      A     I 11.4;
      =     DB3.DBX 220.4;
      A     L 0.0;
      A     I 11.5;
      =     DB3.DBX 1.7;
      A     L 0.0;
      A     I 11.6;
      =     DB3.DBX 220.5;
      A     L 0.0;
      A     I 14.7;
      =     DB3.DBX 254.6;
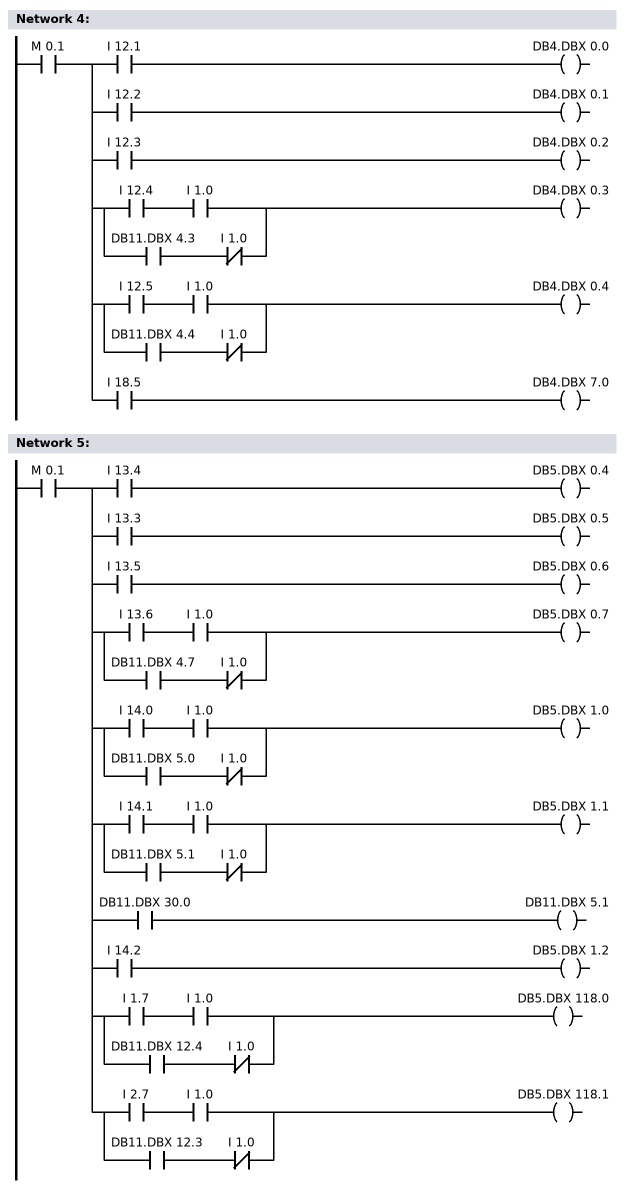
NETWORK
TITLE =
      A     M 0.1;
      =     L 0.0;
      A     L 0.0;
      A     I 12.1;
      =     DB4.DBX 0.0;
      A     L 0.0;
      A     I 12.2;
      =     DB4.DBX 0.1;
      A     L 0.0;
      A     I 12.3;
      =     DB4.DBX 0.2;
      A     L 0.0;
      A(;
      A     I 12.4;
      A     I 1.0;
      O;
      A     DB11.DBX 4.3;
      AN    I 1.0;
      );
      =     DB4.DBX 0.3;
      A     L 0.0;
      A(;
      A     I 12.5;
      A     I 1.0;
      O;
      A     DB11.DBX 4.4;
      AN    I 1.0;
      );
      =     DB4.DBX 0.4;
      A     L 0.0;
      A     I 18.5;
      =     DB4.DBX 7.0;
NETWORK
TITLE =
      A     M 0.1;
      =     L 0.0;
      A     L 0.0;
      A     I 13.4;
      =     DB5.DBX 0.4;
      A     L 0.0;
      A     I 13.3;
      =     DB5.DBX 0.5;
      A     L 0.0;
      A     I 13.5;
      =     DB5.DBX 0.6;
      A     L 0.0;
      A(;
      A     I 13.6;
      A     I 1.0;
      O;
      A     DB11.DBX 4.7;
      AN    I 1.0;
      );
      =     DB5.DBX 0.7;
      A     L 0.0;
      A(;
      A     I 14.0;
      A     I 1.0;
      O;
      A     DB11.DBX 5.0;
      AN    I 1.0;
      );
      =     DB5.DBX 1.0;
      A     L 0.0;
      A(;
      A     I 14.1;
      A     I 1.0;
      O;
      A     DB11.DBX 5.1;
      AN    I 1.0;
      );
      =     DB5.DBX 1.1;
      A     L 0.0;
      A     DB11.DBX 30.0;
      =     DB11.DBX 5.1;
      A     L 0.0;
      A     I 14.2;
      =     DB5.DBX 1.2;
      A     L 0.0;
      A(;
      A     I 1.7;
      A     I 1.0;
      O;
      A     DB11.DBX 12.4;
      AN    I 1.0;
      );
      =     DB5.DBX 118.0;
      A     L 0.0;
      A(;
      A     I 2.7;
      A     I 1.0;
      O;
      A     DB11.DBX 12.3;
      AN    I 1.0;
      );
      =     DB5.DBX 118.1;
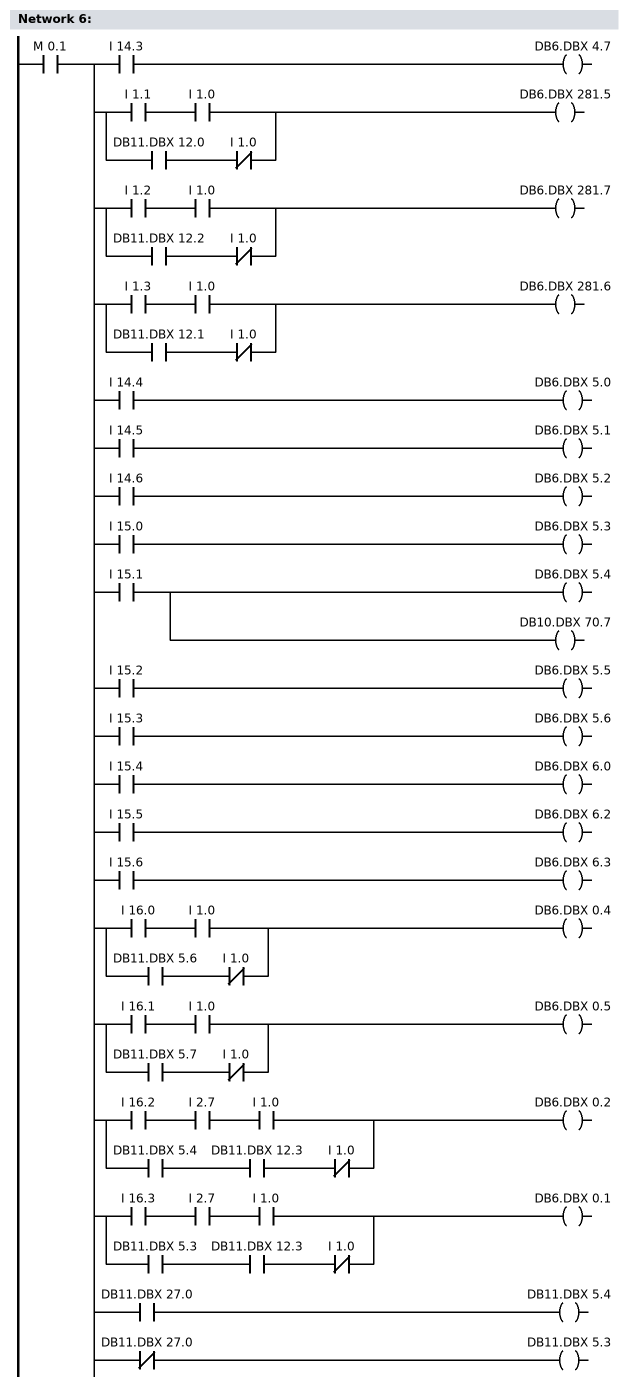
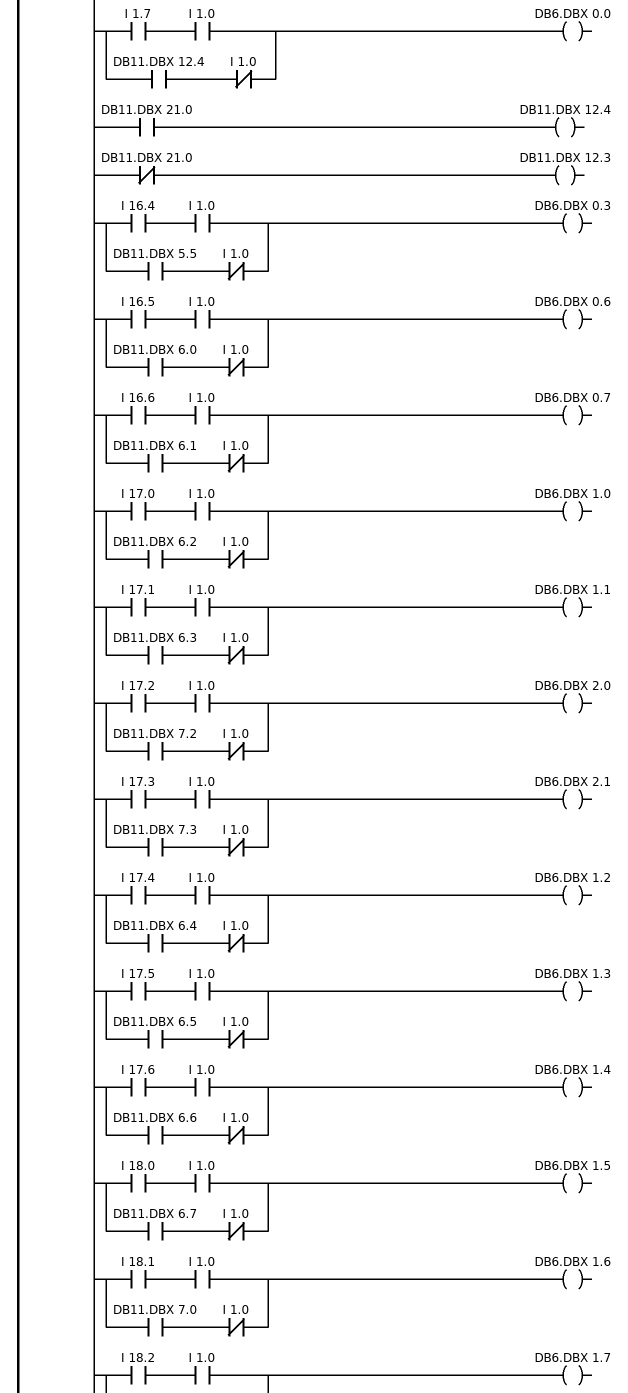
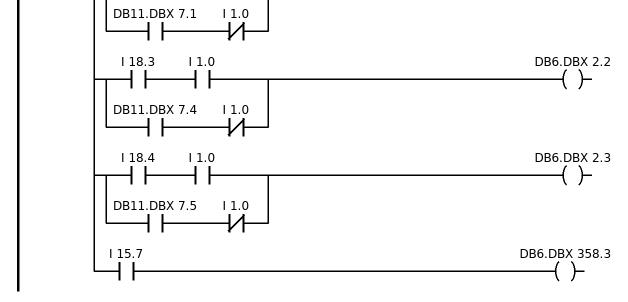
NETWORK
TITLE =
      A     M 0.1;
      =     L 0.0;
      A     L 0.0;
      A     I 14.3;
      =     DB6.DBX 4.7;
      A     L 0.0;
      A(;
      A     I 1.1;
      A     I 1.0;
      O;
      A     DB11.DBX 12.0;
      AN    I 1.0;
      );
      =     DB6.DBX 281.5;
      A     L 0.0;
      A(;
      A     I 1.2;
      A     I 1.0;
      O;
      A     DB11.DBX 12.2;
      AN    I 1.0;
      );
      =     DB6.DBX 281.7;
      A     L 0.0;
      A(;
      A     I 1.3;
      A     I 1.0;
      O;
      A     DB11.DBX 12.1;
      AN    I 1.0;
      );
      =     DB6.DBX 281.6;
      A     L 0.0;
      A     I 14.4;
      =     DB6.DBX 5.0;
      A     L 0.0;
      A     I 14.5;
      =     DB6.DBX 5.1;
      A     L 0.0;
      A     I 14.6;
      =     DB6.DBX 5.2;
      A     L 0.0;
      A     I 15.0;
      =     DB6.DBX 5.3;
      A     L 0.0;
      A     I 15.1;
      =     DB6.DBX 5.4;
      =     DB10.DBX 70.7;
      A     L 0.0;
      A     I 15.2;
      =     DB6.DBX 5.5;
      A     L 0.0;
      A     I 15.3;
      =     DB6.DBX 5.6;
      A     L 0.0;
      A     I 15.4;
      =     DB6.DBX 6.0;
      A     L 0.0;
      A     I 15.5;
      =     DB6.DBX 6.2;
      A     L 0.0;
      A     I 15.6;
      =     DB6.DBX 6.3;
      A     L 0.0;
      A(;
      A     I 16.0;
      A     I 1.0;
      O;
      A     DB11.DBX 5.6;
      AN    I 1.0;
      );
      =     DB6.DBX 0.4;
      A     L 0.0;
      A(;
      A     I 16.1;
      A     I 1.0;
      O;
      A     DB11.DBX 5.7;
      AN    I 1.0;
      );
      =     DB6.DBX 0.5;
      A     L 0.0;
      A(;
      A     I 16.2;
      A     I 2.7;
      A     I 1.0;
      O;
      A     DB11.DBX 5.4;
      A     DB11.DBX 12.3;
      AN    I 1.0;
      );
      =     DB6.DBX 0.2;
      A     L 0.0;
      A(;
      A     I 16.3;
      A     I 2.7;
      A     I 1.0;
      O;
      A     DB11.DBX 5.3;
      A     DB11.DBX 12.3;
      AN    I 1.0;
      );
      =     DB6.DBX 0.1;
      A     L 0.0;
      A     DB11.DBX 27.0;
      =     DB11.DBX 5.4;
      A     L 0.0;
      AN    DB11.DBX 27.0;
      =     DB11.DBX 5.3;
      A     L 0.0;
      A(;
      A     I 1.7;
      A     I 1.0;
      O;
      A     DB11.DBX 12.4;
      AN    I 1.0;
      );
      =     DB6.DBX 0.0;
      A     L 0.0;
      A     DB11.DBX 21.0;
      =     DB11.DBX 12.4;
      A     L 0.0;
      AN    DB11.DBX 21.0;
      =     DB11.DBX 12.3;
      A     L 0.0;
      A(;
      A     I 16.4;
      A     I 1.0;
      O;
      A     DB11.DBX 5.5;
      AN    I 1.0;
      );
      =     DB6.DBX 0.3;
      A     L 0.0;
      A(;
      A     I 16.5;
      A     I 1.0;
      O;
      A     DB11.DBX 6.0;
      AN    I 1.0;
      );
      =     DB6.DBX 0.6;
      A     L 0.0;
      A(;
      A     I 16.6;
      A     I 1.0;
      O;
      A     DB11.DBX 6.1;
      AN    I 1.0;
      );
      =     DB6.DBX 0.7;
      A     L 0.0;
      A(;
      A     I 17.0;
      A     I 1.0;
      O;
      A     DB11.DBX 6.2;
      AN    I 1.0;
      );
      =     DB6.DBX 1.0;
      A     L 0.0;
      A(;
      A     I 17.1;
      A     I 1.0;
      O;
      A     DB11.DBX 6.3;
      AN    I 1.0;
      );
      =     DB6.DBX 1.1;
      A     L 0.0;
      A(;
      A     I 17.2;
      A     I 1.0;
      O;
      A     DB11.DBX 7.2;
      AN    I 1.0;
      );
      =     DB6.DBX 2.0;
      A     L 0.0;
      A(;
      A     I 17.3;
      A     I 1.0;
      O;
      A     DB11.DBX 7.3;
      AN    I 1.0;
      );
      =     DB6.DBX 2.1;
      A     L 0.0;
      A(;
      A     I 17.4;
      A     I 1.0;
      O;
      A     DB11.DBX 6.4;
      AN    I 1.0;
      );
      =     DB6.DBX 1.2;
      A     L 0.0;
      A(;
      A     I 17.5;
      A     I 1.0;
      O;
      A     DB11.DBX 6.5;
      AN    I 1.0;
      );
      =     DB6.DBX 1.3;
      A     L 0.0;
      A(;
      A     I 17.6;
      A     I 1.0;
      O;
      A     DB11.DBX 6.6;
      AN    I 1.0;
      );
      =     DB6.DBX 1.4;
      A     L 0.0;
      A(;
      A     I 18.0;
      A     I 1.0;
      O;
      A     DB11.DBX 6.7;
      AN    I 1.0;
      );
      =     DB6.DBX 1.5;
      A     L 0.0;
      A(;
      A     I 18.1;
      A     I 1.0;
      O;
      A     DB11.DBX 7.0;
      AN    I 1.0;
      );
      =     DB6.DBX 1.6;
      A     L 0.0;
      A(;
      A     I 18.2;
      A     I 1.0;
      O;
      A     DB11.DBX 7.1;
      AN    I 1.0;
      );
      =     DB6.DBX 1.7;
      A     L 0.0;
      A(;
      A     I 18.3;
      A     I 1.0;
      O;
      A     DB11.DBX 7.4;
      AN    I 1.0;
      );
      =     DB6.DBX 2.2;
      A     L 0.0;
      A(;
      A     I 18.4;
      A     I 1.0;
      O;
      A     DB11.DBX 7.5;
      AN    I 1.0;
      );
      =     DB6.DBX 2.3;
      A     L 0.0;
      A     I 15.7;
      =     DB6.DBX 358.3;
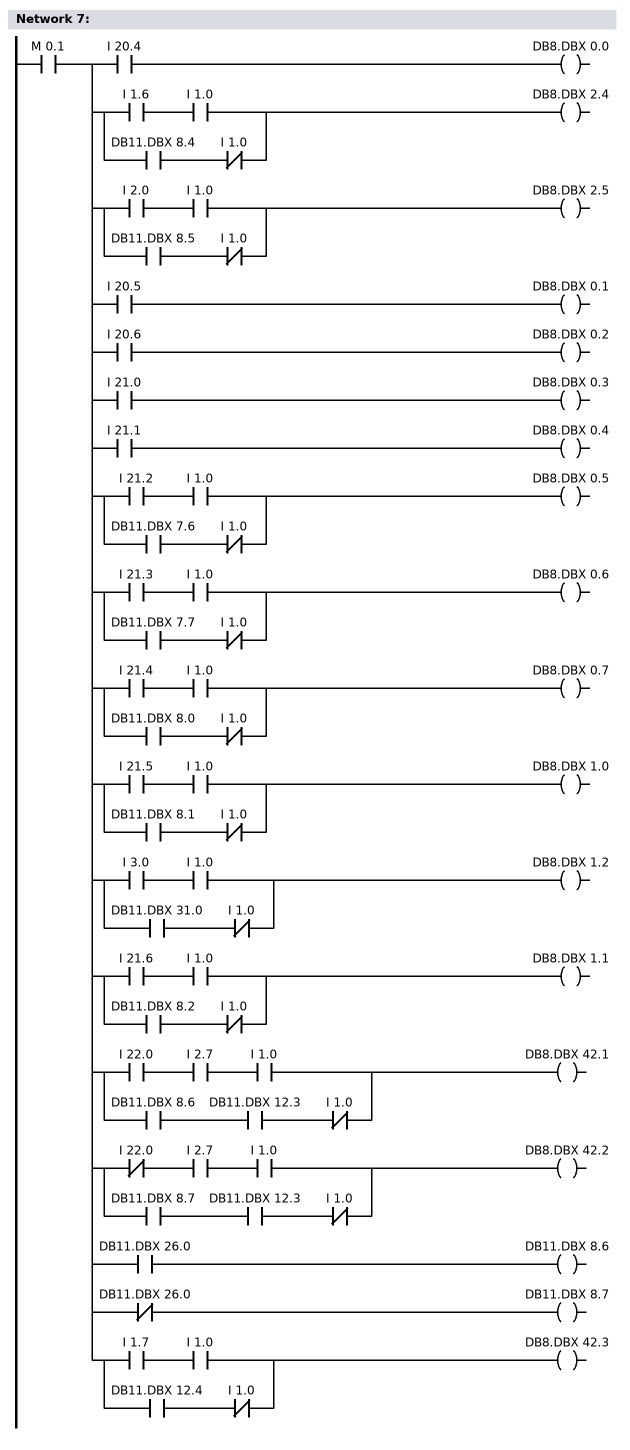
NETWORK
TITLE =
      A     M 0.1;
      =     L 0.0;
      A     L 0.0;
      A     I 20.4;
      =     DB8.DBX 0.0;
      A     L 0.0;
      A(;
      A     I 1.6;
      A     I 1.0;
      O;
      A     DB11.DBX 8.4;
      AN    I 1.0;
      );
      =     DB8.DBX 2.4;
      A     L 0.0;
      A(;
      A     I 2.0;
      A     I 1.0;
      O;
      A     DB11.DBX 8.5;
      AN    I 1.0;
      );
      =     DB8.DBX 2.5;
      A     L 0.0;
      A     I 20.5;
      =     DB8.DBX 0.1;
      A     L 0.0;
      A     I 20.6;
      =     DB8.DBX 0.2;
      A     L 0.0;
      A     I 21.0;
      =     DB8.DBX 0.3;
      A     L 0.0;
      A     I 21.1;
      =     DB8.DBX 0.4;
      A     L 0.0;
      A(;
      A     I 21.2;
      A     I 1.0;
      O;
      A     DB11.DBX 7.6;
      AN    I 1.0;
      );
      =     DB8.DBX 0.5;
      A     L 0.0;
      A(;
      A     I 21.3;
      A     I 1.0;
      O;
      A     DB11.DBX 7.7;
      AN    I 1.0;
      );
      =     DB8.DBX 0.6;
      A     L 0.0;
      A(;
      A     I 21.4;
      A     I 1.0;
      O;
      A     DB11.DBX 8.0;
      AN    I 1.0;
      );
      =     DB8.DBX 0.7;
      A     L 0.0;
      A(;
      A     I 21.5;
      A     I 1.0;
      O;
      A     DB11.DBX 8.1;
      AN    I 1.0;
      );
      =     DB8.DBX 1.0;
      A     L 0.0;
      A(;
      A     I 3.0;
      A     I 1.0;
      O;
      A     DB11.DBX 31.0;
      AN    I 1.0;
      );
      =     DB8.DBX 1.2;
      A     L 0.0;
      A(;
      A     I 21.6;
      A     I 1.0;
      O;
      A     DB11.DBX 8.2;
      AN    I 1.0;
      );
      =     DB8.DBX 1.1;
      A     L 0.0;
      A(;
      A     I 22.0;
      A     I 2.7;
      A     I 1.0;
      O;
      A     DB11.DBX 8.6;
      A     DB11.DBX 12.3;
      AN    I 1.0;
      );
      =     DB8.DBX 42.1;
      A     L 0.0;
      A(;
      AN    I 22.0;
      A     I 2.7;
      A     I 1.0;
      O;
      A     DB11.DBX 8.7;
      A     DB11.DBX 12.3;
      AN    I 1.0;
      );
      =     DB8.DBX 42.2;
      A     L 0.0;
      A     DB11.DBX 26.0;
      =     DB11.DBX 8.6;
      A     L 0.0;
      AN    DB11.DBX 26.0;
      =     DB11.DBX 8.7;
      A     L 0.0;
      A(;
      A     I 1.7;
      A     I 1.0;
      O;
      A     DB11.DBX 12.4;
      AN    I 1.0;
      );
      =     DB8.DBX 42.3;
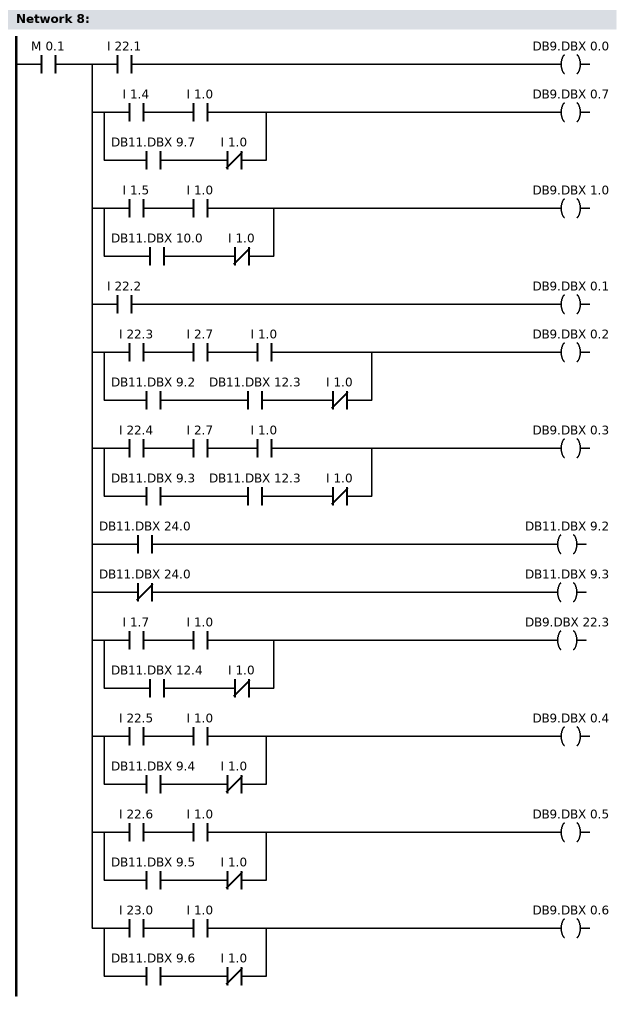
NETWORK
TITLE =
      A     M 0.1;
      =     L 0.0;
      A     L 0.0;
      A     I 22.1;
      =     DB9.DBX 0.0;
      A     L 0.0;
      A(;
      A     I 1.4;
      A     I 1.0;
      O;
      A     DB11.DBX 9.7;
      AN    I 1.0;
      );
      =     DB9.DBX 0.7;
      A     L 0.0;
      A(;
      A     I 1.5;
      A     I 1.0;
      O;
      A     DB11.DBX 10.0;
      AN    I 1.0;
      );
      =     DB9.DBX 1.0;
      A     L 0.0;
      A     I 22.2;
      =     DB9.DBX 0.1;
      A     L 0.0;
      A(;
      A     I 22.3;
      A     I 2.7;
      A     I 1.0;
      O;
      A     DB11.DBX 9.2;
      A     DB11.DBX 12.3;
      AN    I 1.0;
      );
      =     DB9.DBX 0.2;
      A     L 0.0;
      A(;
      A     I 22.4;
      A     I 2.7;
      A     I 1.0;
      O;
      A     DB11.DBX 9.3;
      A     DB11.DBX 12.3;
      AN    I 1.0;
      );
      =     DB9.DBX 0.3;
      A     L 0.0;
      A     DB11.DBX 24.0;
      =     DB11.DBX 9.2;
      A     L 0.0;
      AN    DB11.DBX 24.0;
      =     DB11.DBX 9.3;
      A     L 0.0;
      A(;
      A     I 1.7;
      A     I 1.0;
      O;
      A     DB11.DBX 12.4;
      AN    I 1.0;
      );
      =     DB9.DBX 22.3;
      A     L 0.0;
      A(;
      A     I 22.5;
      A     I 1.0;
      O;
      A     DB11.DBX 9.4;
      AN    I 1.0;
      );
      =     DB9.DBX 0.4;
      A     L 0.0;
      A(;
      A     I 22.6;
      A     I 1.0;
      O;
      A     DB11.DBX 9.5;
      AN    I 1.0;
      );
      =     DB9.DBX 0.5;
      A     L 0.0;
      A(;
      A     I 23.0;
      A     I 1.0;
      O;
      A     DB11.DBX 9.6;
      AN    I 1.0;
      );
      =     DB9.DBX 0.6;
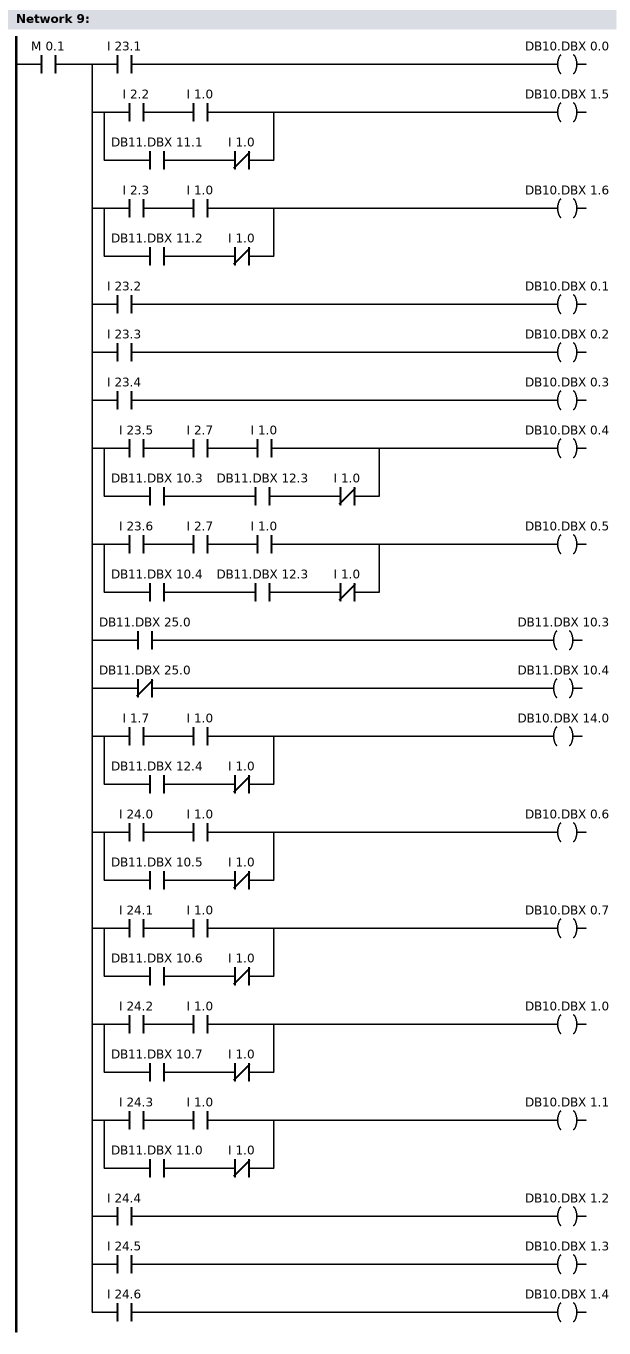
NETWORK
TITLE =
      A     M 0.1;
      =     L 0.0;
      A     L 0.0;
      A     I 23.1;
      =     DB10.DBX 0.0;
      A     L 0.0;
      A(;
      A     I 2.2;
      A     I 1.0;
      O;
      A     DB11.DBX 11.1;
      AN    I 1.0;
      );
      =     DB10.DBX 1.5;
      A     L 0.0;
      A(;
      A     I 2.3;
      A     I 1.0;
      O;
      A     DB11.DBX 11.2;
      AN    I 1.0;
      );
      =     DB10.DBX 1.6;
      A     L 0.0;
      A     I 23.2;
      =     DB10.DBX 0.1;
      A     L 0.0;
      A     I 23.3;
      =     DB10.DBX 0.2;
      A     L 0.0;
      A     I 23.4;
      =     DB10.DBX 0.3;
      A     L 0.0;
      A(;
      A     I 23.5;
      A     I 2.7;
      A     I 1.0;
      O;
      A     DB11.DBX 10.3;
      A     DB11.DBX 12.3;
      AN    I 1.0;
      );
      =     DB10.DBX 0.4;
      A     L 0.0;
      A(;
      A     I 23.6;
      A     I 2.7;
      A     I 1.0;
      O;
      A     DB11.DBX 10.4;
      A     DB11.DBX 12.3;
      AN    I 1.0;
      );
      =     DB10.DBX 0.5;
      A     L 0.0;
      A     DB11.DBX 25.0;
      =     DB11.DBX 10.3;
      A     L 0.0;
      AN    DB11.DBX 25.0;
      =     DB11.DBX 10.4;
      A     L 0.0;
      A(;
      A     I 1.7;
      A     I 1.0;
      O;
      A     DB11.DBX 12.4;
      AN    I 1.0;
      );
      =     DB10.DBX 14.0;
      A     L 0.0;
      A(;
      A     I 24.0;
      A     I 1.0;
      O;
      A     DB11.DBX 10.5;
      AN    I 1.0;
      );
      =     DB10.DBX 0.6;
      A     L 0.0;
      A(;
      A     I 24.1;
      A     I 1.0;
      O;
      A     DB11.DBX 10.6;
      AN    I 1.0;
      );
      =     DB10.DBX 0.7;
      A     L 0.0;
      A(;
      A     I 24.2;
      A     I 1.0;
      O;
      A     DB11.DBX 10.7;
      AN    I 1.0;
      );
      =     DB10.DBX 1.0;
      A     L 0.0;
      A(;
      A     I 24.3;
      A     I 1.0;
      O;
      A     DB11.DBX 11.0;
      AN    I 1.0;
      );
      =     DB10.DBX 1.1;
      A     L 0.0;
      A     I 24.4;
      =     DB10.DBX 1.2;
      A     L 0.0;
      A     I 24.5;
      =     DB10.DBX 1.3;
      A     L 0.0;
      A     I 24.6;
      =     DB10.DBX 1.4;
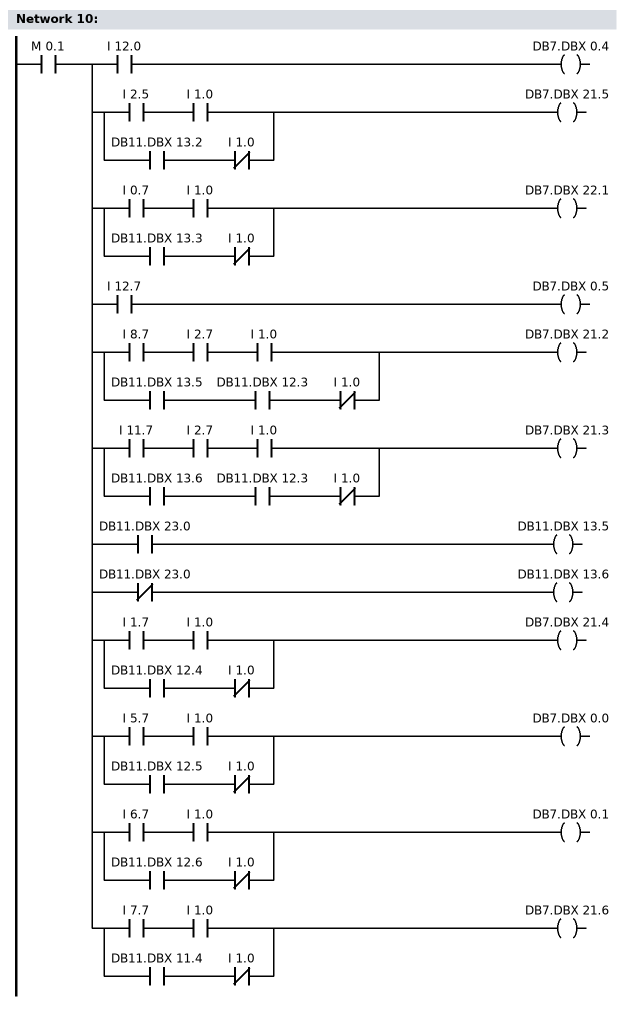
NETWORK
TITLE =
      A     M 0.1;
      =     L 0.0;
      A     L 0.0;
      A     I 12.0;
      =     DB7.DBX 0.4;
      A     L 0.0;
      A(;
      A     I 2.5;
      A     I 1.0;
      O;
      A     DB11.DBX 13.2;
      AN    I 1.0;
      );
      =     DB7.DBX 21.5;
      A     L 0.0;
      A(;
      A     I 0.7;
      A     I 1.0;
      O;
      A     DB11.DBX 13.3;
      AN    I 1.0;
      );
      =     DB7.DBX 22.1;
      A     L 0.0;
      A     I 12.7;
      =     DB7.DBX 0.5;
      A     L 0.0;
      A(;
      A     I 8.7;
      A     I 2.7;
      A     I 1.0;
      O;
      A     DB11.DBX 13.5;
      A     DB11.DBX 12.3;
      AN    I 1.0;
      );
      =     DB7.DBX 21.2;
      A     L 0.0;
      A(;
      A     I 11.7;
      A     I 2.7;
      A     I 1.0;
      O;
      A     DB11.DBX 13.6;
      A     DB11.DBX 12.3;
      AN    I 1.0;
      );
      =     DB7.DBX 21.3;
      A     L 0.0;
      A     DB11.DBX 23.0;
      =     DB11.DBX 13.5;
      A     L 0.0;
      AN    DB11.DBX 23.0;
      =     DB11.DBX 13.6;
      A     L 0.0;
      A(;
      A     I 1.7;
      A     I 1.0;
      O;
      A     DB11.DBX 12.4;
      AN    I 1.0;
      );
      =     DB7.DBX 21.4;
      A     L 0.0;
      A(;
      A     I 5.7;
      A     I 1.0;
      O;
      A     DB11.DBX 12.5;
      AN    I 1.0;
      );
      =     DB7.DBX 0.0;
      A     L 0.0;
      A(;
      A     I 6.7;
      A     I 1.0;
      O;
      A     DB11.DBX 12.6;
      AN    I 1.0;
      );
      =     DB7.DBX 0.1;
      A     L 0.0;
      A(;
      A     I 7.7;
      A     I 1.0;
      O;
      A     DB11.DBX 11.4;
      AN    I 1.0;
      );
      =     DB7.DBX 21.6;
END_FUNCTION

FUNCTION FC 2 : VOID
AUTHOR : Kamillas
VERSION : 0.1
BEGIN
// (block stored without names or comments; labels and parameter names are numbered)
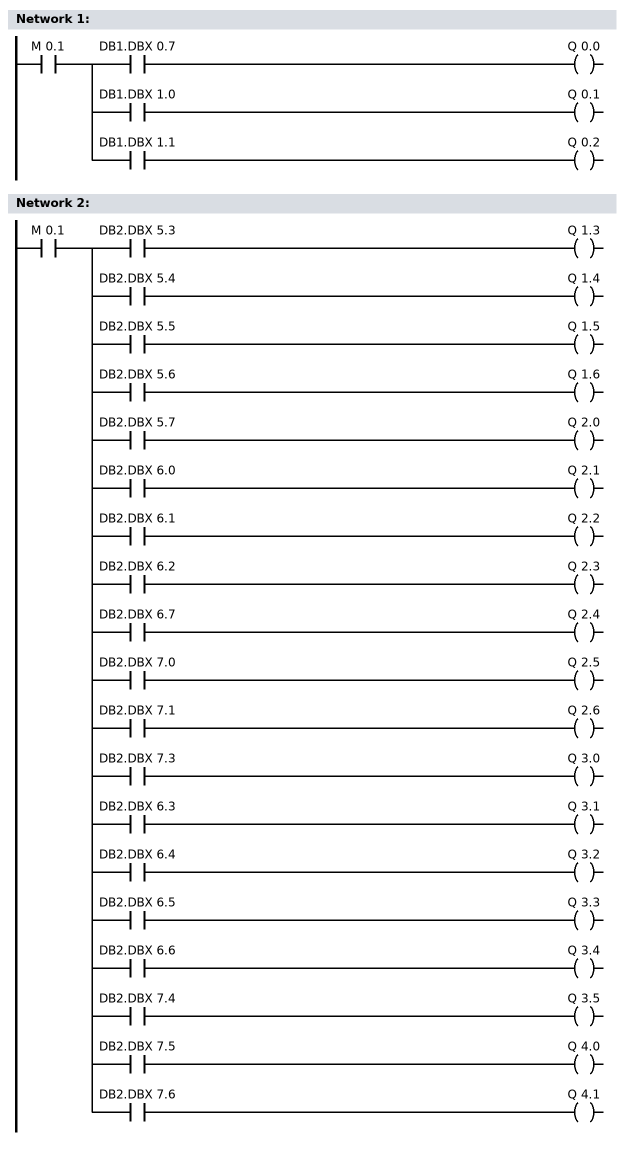
NETWORK
TITLE =
      A     M 0.1;
      =     L 0.0;
      A     L 0.0;
      A     DB1.DBX 0.7;
      =     Q 0.0;
      A     L 0.0;
      A     DB1.DBX 1.0;
      =     Q 0.1;
      A     L 0.0;
      A     DB1.DBX 1.1;
      =     Q 0.2;
NETWORK
TITLE =
      A     M 0.1;
      =     L 0.0;
      A     L 0.0;
      A     DB2.DBX 5.3;
      =     Q 1.3;
      A     L 0.0;
      A     DB2.DBX 5.4;
      =     Q 1.4;
      A     L 0.0;
      A     DB2.DBX 5.5;
      =     Q 1.5;
      A     L 0.0;
      A     DB2.DBX 5.6;
      =     Q 1.6;
      A     L 0.0;
      A     DB2.DBX 5.7;
      =     Q 2.0;
      A     L 0.0;
      A     DB2.DBX 6.0;
      =     Q 2.1;
      A     L 0.0;
      A     DB2.DBX 6.1;
      =     Q 2.2;
      A     L 0.0;
      A     DB2.DBX 6.2;
      =     Q 2.3;
      A     L 0.0;
      A     DB2.DBX 6.7;
      =     Q 2.4;
      A     L 0.0;
      A     DB2.DBX 7.0;
      =     Q 2.5;
      A     L 0.0;
      A     DB2.DBX 7.1;
      =     Q 2.6;
      A     L 0.0;
      A     DB2.DBX 7.3;
      =     Q 3.0;
      A     L 0.0;
      A     DB2.DBX 6.3;
      =     Q 3.1;
      A     L 0.0;
      A     DB2.DBX 6.4;
      =     Q 3.2;
      A     L 0.0;
      A     DB2.DBX 6.5;
      =     Q 3.3;
      A     L 0.0;
      A     DB2.DBX 6.6;
      =     Q 3.4;
      A     L 0.0;
      A     DB2.DBX 7.4;
      =     Q 3.5;
      A     L 0.0;
      A     DB2.DBX 7.5;
      =     Q 4.0;
      A     L 0.0;
      A     DB2.DBX 7.6;
      =     Q 4.1;
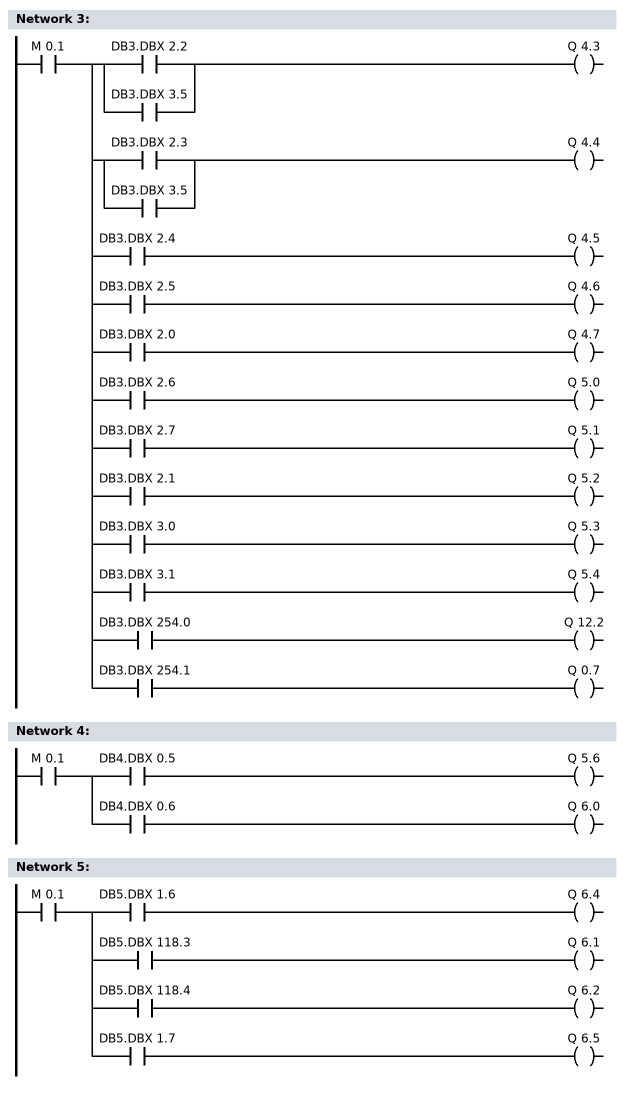
NETWORK
TITLE =
      A     M 0.1;
      =     L 0.0;
      A     L 0.0;
      A(;
      O     DB3.DBX 2.2;
      O     DB3.DBX 3.5;
      );
      =     Q 4.3;
      A     L 0.0;
      A(;
      O     DB3.DBX 2.3;
      O     DB3.DBX 3.5;
      );
      =     Q 4.4;
      A     L 0.0;
      A     DB3.DBX 2.4;
      =     Q 4.5;
      A     L 0.0;
      A     DB3.DBX 2.5;
      =     Q 4.6;
      A     L 0.0;
      A     DB3.DBX 2.0;
      =     Q 4.7;
      A     L 0.0;
      A     DB3.DBX 2.6;
      =     Q 5.0;
      A     L 0.0;
      A     DB3.DBX 2.7;
      =     Q 5.1;
      A     L 0.0;
      A     DB3.DBX 2.1;
      =     Q 5.2;
      A     L 0.0;
      A     DB3.DBX 3.0;
      =     Q 5.3;
      A     L 0.0;
      A     DB3.DBX 3.1;
      =     Q 5.4;
      A     L 0.0;
      A     DB3.DBX 254.0;
      =     Q 12.2;
      A     L 0.0;
      A     DB3.DBX 254.1;
      =     Q 0.7;
NETWORK
TITLE =
      A     M 0.1;
      =     L 0.0;
      A     L 0.0;
      A     DB4.DBX 0.5;
      =     Q 5.6;
      A     L 0.0;
      A     DB4.DBX 0.6;
      =     Q 6.0;
NETWORK
TITLE =
      A     M 0.1;
      =     L 0.0;
      A     L 0.0;
      A     DB5.DBX 1.6;
      =     Q 6.4;
      A     L 0.0;
      A     DB5.DBX 118.3;
      =     Q 6.1;
      A     L 0.0;
      A     DB5.DBX 118.4;
      =     Q 6.2;
      A     L 0.0;
      A     DB5.DBX 1.7;
      =     Q 6.5;
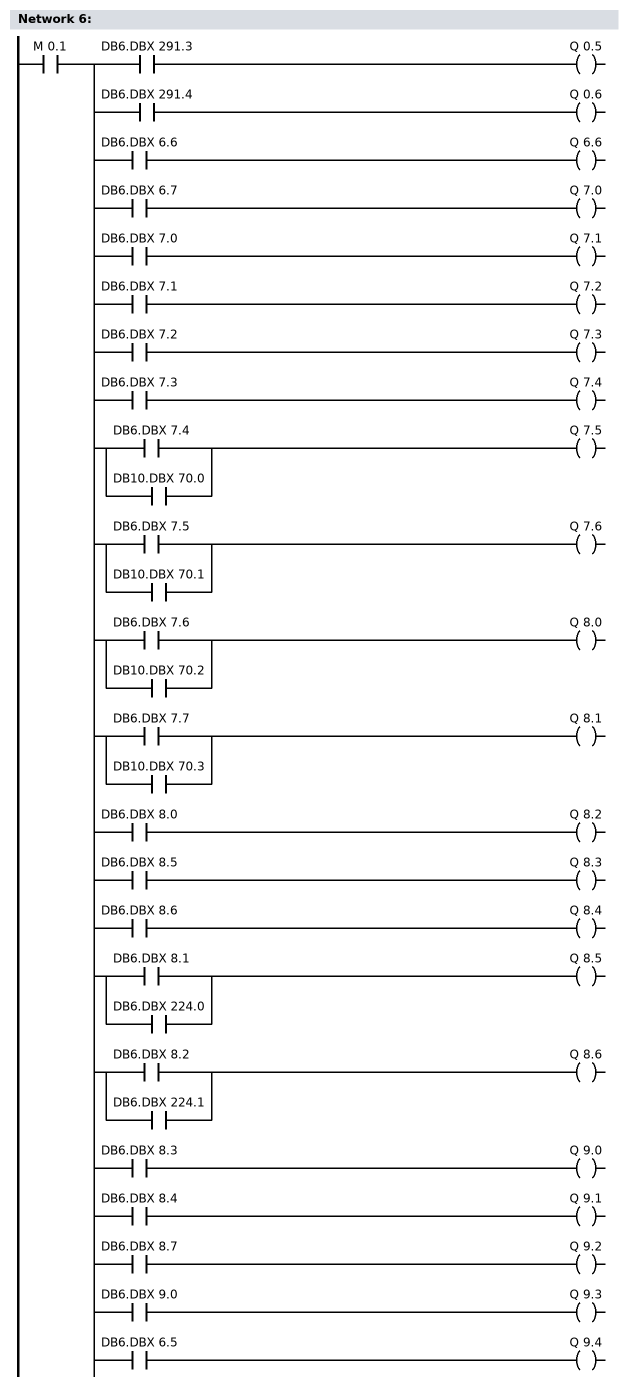
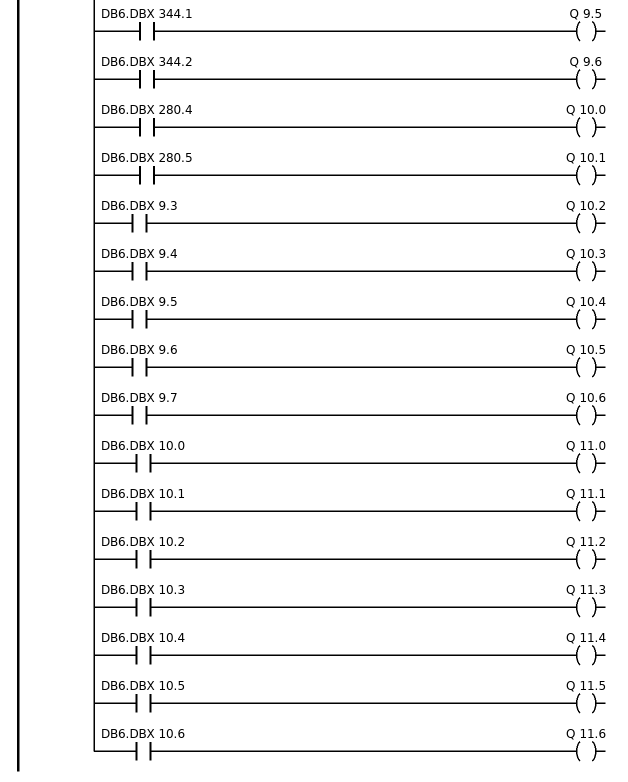
NETWORK
TITLE =
      A     M 0.1;
      =     L 0.0;
      A     L 0.0;
      A     DB6.DBX 291.3;
      =     Q 0.5;
      A     L 0.0;
      A     DB6.DBX 291.4;
      =     Q 0.6;
      A     L 0.0;
      A     DB6.DBX 6.6;
      =     Q 6.6;
      A     L 0.0;
      A     DB6.DBX 6.7;
      =     Q 7.0;
      A     L 0.0;
      A     DB6.DBX 7.0;
      =     Q 7.1;
      A     L 0.0;
      A     DB6.DBX 7.1;
      =     Q 7.2;
      A     L 0.0;
      A     DB6.DBX 7.2;
      =     Q 7.3;
      A     L 0.0;
      A     DB6.DBX 7.3;
      =     Q 7.4;
      A     L 0.0;
      A(;
      O     DB6.DBX 7.4;
      O     DB10.DBX 70.0;
      );
      =     Q 7.5;
      A     L 0.0;
      A(;
      O     DB6.DBX 7.5;
      O     DB10.DBX 70.1;
      );
      =     Q 7.6;
      A     L 0.0;
      A(;
      O     DB6.DBX 7.6;
      O     DB10.DBX 70.2;
      );
      =     Q 8.0;
      A     L 0.0;
      A(;
      O     DB6.DBX 7.7;
      O     DB10.DBX 70.3;
      );
      =     Q 8.1;
      A     L 0.0;
      A     DB6.DBX 8.0;
      =     Q 8.2;
      A     L 0.0;
      A     DB6.DBX 8.5;
      =     Q 8.3;
      A     L 0.0;
      A     DB6.DBX 8.6;
      =     Q 8.4;
      A     L 0.0;
      A(;
      O     DB6.DBX 8.1;
      O     DB6.DBX 224.0;
      );
      =     Q 8.5;
      A     L 0.0;
      A(;
      O     DB6.DBX 8.2;
      O     DB6.DBX 224.1;
      );
      =     Q 8.6;
      A     L 0.0;
      A     DB6.DBX 8.3;
      =     Q 9.0;
      A     L 0.0;
      A     DB6.DBX 8.4;
      =     Q 9.1;
      A     L 0.0;
      A     DB6.DBX 8.7;
      =     Q 9.2;
      A     L 0.0;
      A     DB6.DBX 9.0;
      =     Q 9.3;
      A     L 0.0;
      A     DB6.DBX 6.5;
      =     Q 9.4;
      A     L 0.0;
      A     DB6.DBX 344.1;
      =     Q 9.5;
      A     L 0.0;
      A     DB6.DBX 344.2;
      =     Q 9.6;
      A     L 0.0;
      A     DB6.DBX 280.4;
      =     Q 10.0;
      A     L 0.0;
      A     DB6.DBX 280.5;
      =     Q 10.1;
      A     L 0.0;
      A     DB6.DBX 9.3;
      =     Q 10.2;
      A     L 0.0;
      A     DB6.DBX 9.4;
      =     Q 10.3;
      A     L 0.0;
      A     DB6.DBX 9.5;
      =     Q 10.4;
      A     L 0.0;
      A     DB6.DBX 9.6;
      =     Q 10.5;
      A     L 0.0;
      A     DB6.DBX 9.7;
      =     Q 10.6;
      A     L 0.0;
      A     DB6.DBX 10.0;
      =     Q 11.0;
      A     L 0.0;
      A     DB6.DBX 10.1;
      =     Q 11.1;
      A     L 0.0;
      A     DB6.DBX 10.2;
      =     Q 11.2;
      A     L 0.0;
      A     DB6.DBX 10.3;
      =     Q 11.3;
      A     L 0.0;
      A     DB6.DBX 10.4;
      =     Q 11.4;
      A     L 0.0;
      A     DB6.DBX 10.5;
      =     Q 11.5;
      A     L 0.0;
      A     DB6.DBX 10.6;
      =     Q 11.6;
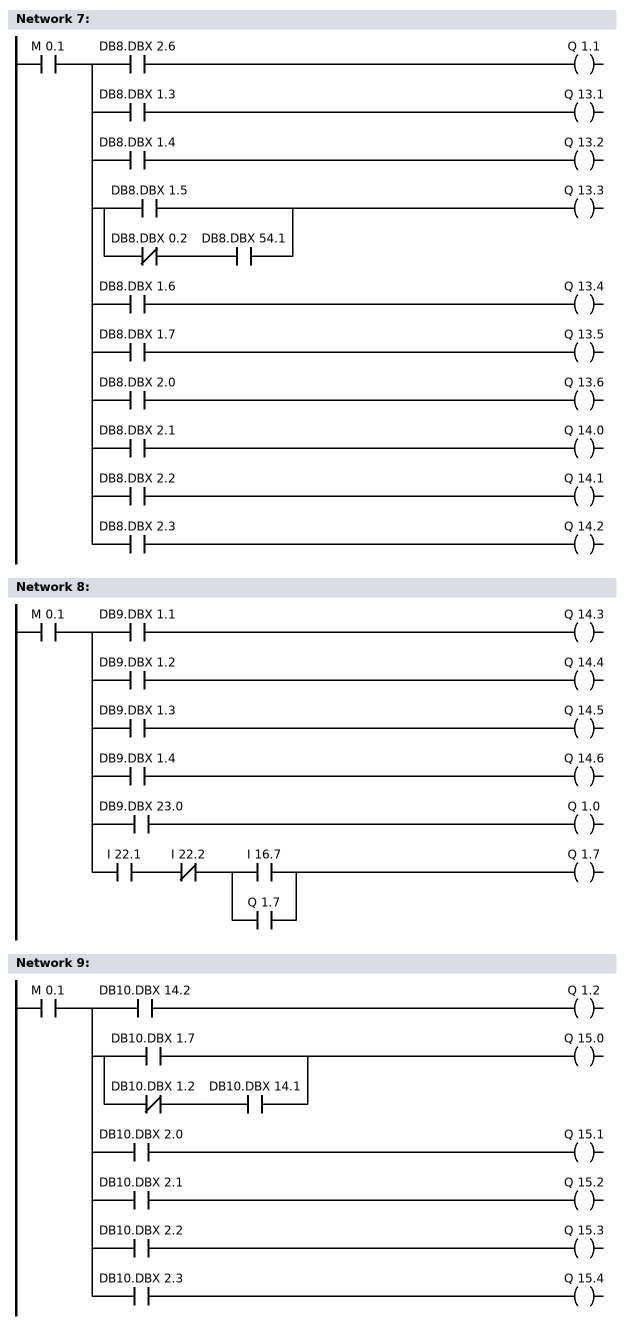
NETWORK
TITLE =
      A     M 0.1;
      =     L 0.0;
      A     L 0.0;
      A     DB8.DBX 2.6;
      =     Q 1.1;
      A     L 0.0;
      A     DB8.DBX 1.3;
      =     Q 13.1;
      A     L 0.0;
      A     DB8.DBX 1.4;
      =     Q 13.2;
      A     L 0.0;
      A(;
      O     DB8.DBX 1.5;
      O;
      AN    DB8.DBX 0.2;
      A     DB8.DBX 54.1;
      );
      =     Q 13.3;
      A     L 0.0;
      A     DB8.DBX 1.6;
      =     Q 13.4;
      A     L 0.0;
      A     DB8.DBX 1.7;
      =     Q 13.5;
      A     L 0.0;
      A     DB8.DBX 2.0;
      =     Q 13.6;
      A     L 0.0;
      A     DB8.DBX 2.1;
      =     Q 14.0;
      A     L 0.0;
      A     DB8.DBX 2.2;
      =     Q 14.1;
      A     L 0.0;
      A     DB8.DBX 2.3;
      =     Q 14.2;
NETWORK
TITLE =
      A     M 0.1;
      =     L 0.0;
      A     L 0.0;
      A     DB9.DBX 1.1;
      =     Q 14.3;
      A     L 0.0;
      A     DB9.DBX 1.2;
      =     Q 14.4;
      A     L 0.0;
      A     DB9.DBX 1.3;
      =     Q 14.5;
      A     L 0.0;
      A     DB9.DBX 1.4;
      =     Q 14.6;
      A     L 0.0;
      A     DB9.DBX 23.0;
      =     Q 1.0;
      A     L 0.0;
      A     I 22.1;
      AN    I 22.2;
      A(;
      O     I 16.7;
      O     Q 1.7;
      );
      =     Q 1.7;
NETWORK
TITLE =
      A     M 0.1;
      =     L 0.0;
      A     L 0.0;
      A     DB10.DBX 14.2;
      =     Q 1.2;
      A     L 0.0;
      A(;
      O     DB10.DBX 1.7;
      O;
      AN    DB10.DBX 1.2;
      A     DB10.DBX 14.1;
      );
      =     Q 15.0;
      A     L 0.0;
      A     DB10.DBX 2.0;
      =     Q 15.1;
      A     L 0.0;
      A     DB10.DBX 2.1;
      =     Q 15.2;
      A     L 0.0;
      A     DB10.DBX 2.2;
      =     Q 15.3;
      A     L 0.0;
      A     DB10.DBX 2.3;
      =     Q 15.4;
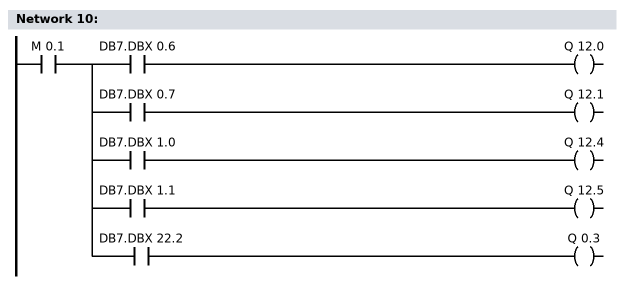
NETWORK
TITLE =
      A     M 0.1;
      =     L 0.0;
      A     L 0.0;
      A     DB7.DBX 0.6;
      =     Q 12.0;
      A     L 0.0;
      A     DB7.DBX 0.7;
      =     Q 12.1;
      A     L 0.0;
      A     DB7.DBX 1.0;
      =     Q 12.4;
      A     L 0.0;
      A     DB7.DBX 1.1;
      =     Q 12.5;
      A     L 0.0;
      A     DB7.DBX 22.2;
      =     Q 0.3;
END_FUNCTION

FUNCTION FC 3 : VOID
AUTHOR : Kamillas
VERSION : 0.1
BEGIN
// (block stored without names or comments; labels and parameter names are numbered)
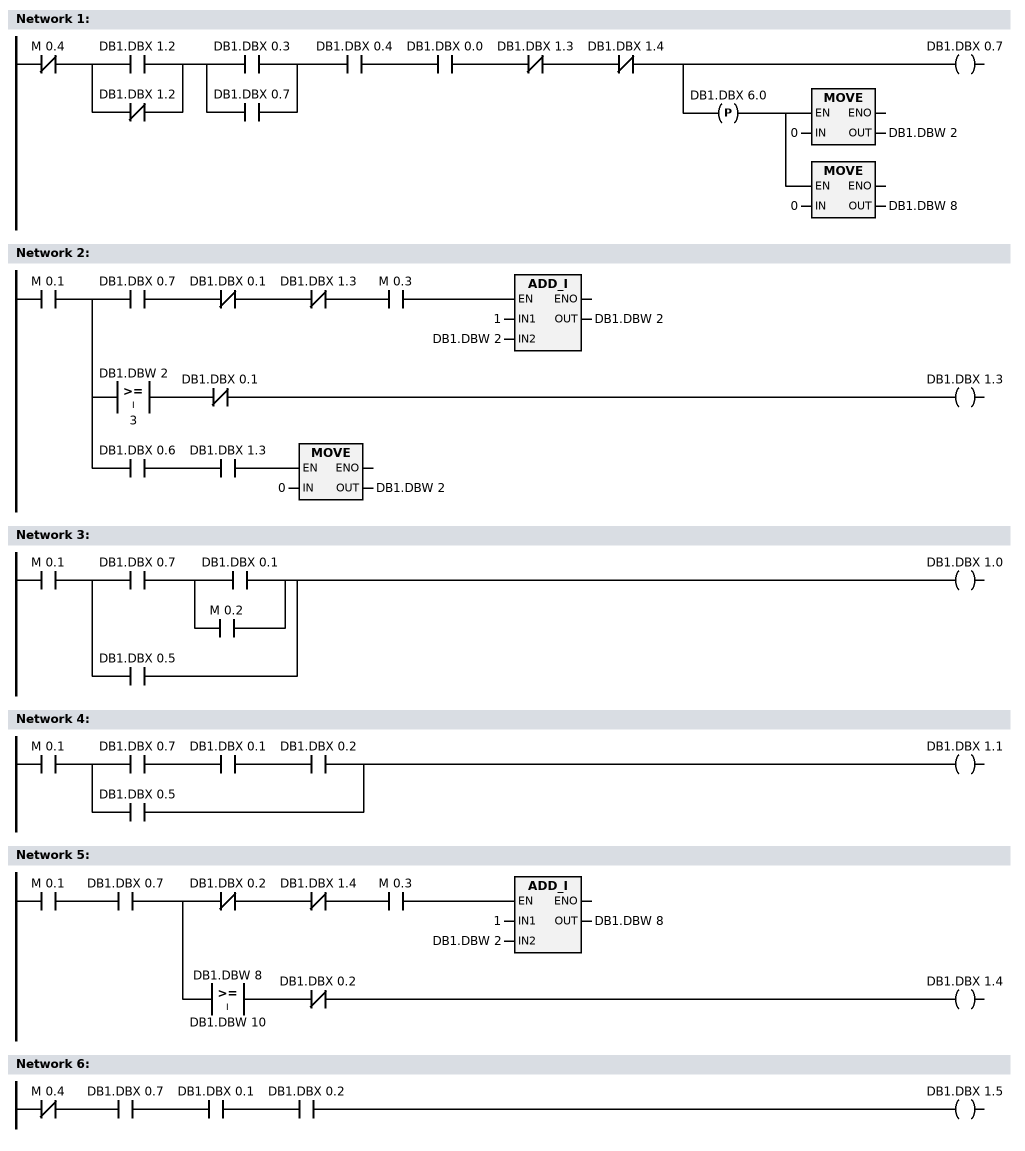
NETWORK
TITLE =
      AN    M 0.4;
      A(;
      O     DB1.DBX 1.2;
      ON    DB1.DBX 1.2;
      );
      A(;
      O     DB1.DBX 0.3;
      O     DB1.DBX 0.7;
      );
      A     DB1.DBX 0.4;
      A     DB1.DBX 0.0;
      AN    DB1.DBX 1.3;
      AN    DB1.DBX 1.4;
      =     L 0.0;
      A     L 0.0;
      BLD   102;
      =     DB1.DBX 0.7;
      A     L 0.0;
      FP    DB1.DBX 6.0;
      =     L 0.1;
      A     L 0.1;
      JNB   M001;
      L     0;
      T     DB1.DBW 2;
M001: NOP   0;
      A     L 0.1;
      JNB   M002;
      L     0;
      T     DB1.DBW 8;
M002: NOP   0;
NETWORK
TITLE =
      A     M 0.1;
      =     L 0.0;
      A     L 0.0;
      A     DB1.DBX 0.7;
      AN    DB1.DBX 0.1;
      AN    DB1.DBX 1.3;
      A     M 0.3;
      JNB   M003;
      L     1;
      L     DB1.DBW 2;
      +I;
      T     DB1.DBW 2;
M003: NOP   0;
      A     L 0.0;
      A(;
      L     DB1.DBW 2;
      L     3;
      >=I;
      );
      AN    DB1.DBX 0.1;
      =     DB1.DBX 1.3;
      A     L 0.0;
      A     DB1.DBX 0.6;
      A     DB1.DBX 1.3;
      JNB   M004;
      L     0;
      T     DB1.DBW 2;
M004: NOP   0;
NETWORK
TITLE =
      A     M 0.1;
      A(;
      A     DB1.DBX 0.7;
      A(;
      O     DB1.DBX 0.1;
      O     M 0.2;
      );
      O     DB1.DBX 0.5;
      );
      =     DB1.DBX 1.0;
NETWORK
TITLE =
      A     M 0.1;
      A(;
      A     DB1.DBX 0.7;
      A     DB1.DBX 0.1;
      A     DB1.DBX 0.2;
      O     DB1.DBX 0.5;
      );
      =     DB1.DBX 1.1;
NETWORK
TITLE =
      A     M 0.1;
      A     DB1.DBX 0.7;
      =     L 0.0;
      A     L 0.0;
      AN    DB1.DBX 0.2;
      AN    DB1.DBX 1.4;
      A     M 0.3;
      JNB   M005;
      L     1;
      L     DB1.DBW 2;
      +I;
      T     DB1.DBW 8;
M005: NOP   0;
      A     L 0.0;
      A(;
      L     DB1.DBW 8;
      L     DB1.DBW 10;
      >=I;
      );
      AN    DB1.DBX 0.2;
      =     DB1.DBX 1.4;
NETWORK
TITLE =
      AN    M 0.4;
      A     DB1.DBX 0.7;
      A     DB1.DBX 0.1;
      A     DB1.DBX 0.2;
      =     DB1.DBX 1.5;
END_FUNCTION

FUNCTION FC 4 : VOID
AUTHOR : Kamillas
VERSION : 0.1
BEGIN
// (block stored without names or comments; labels and parameter names are numbered)
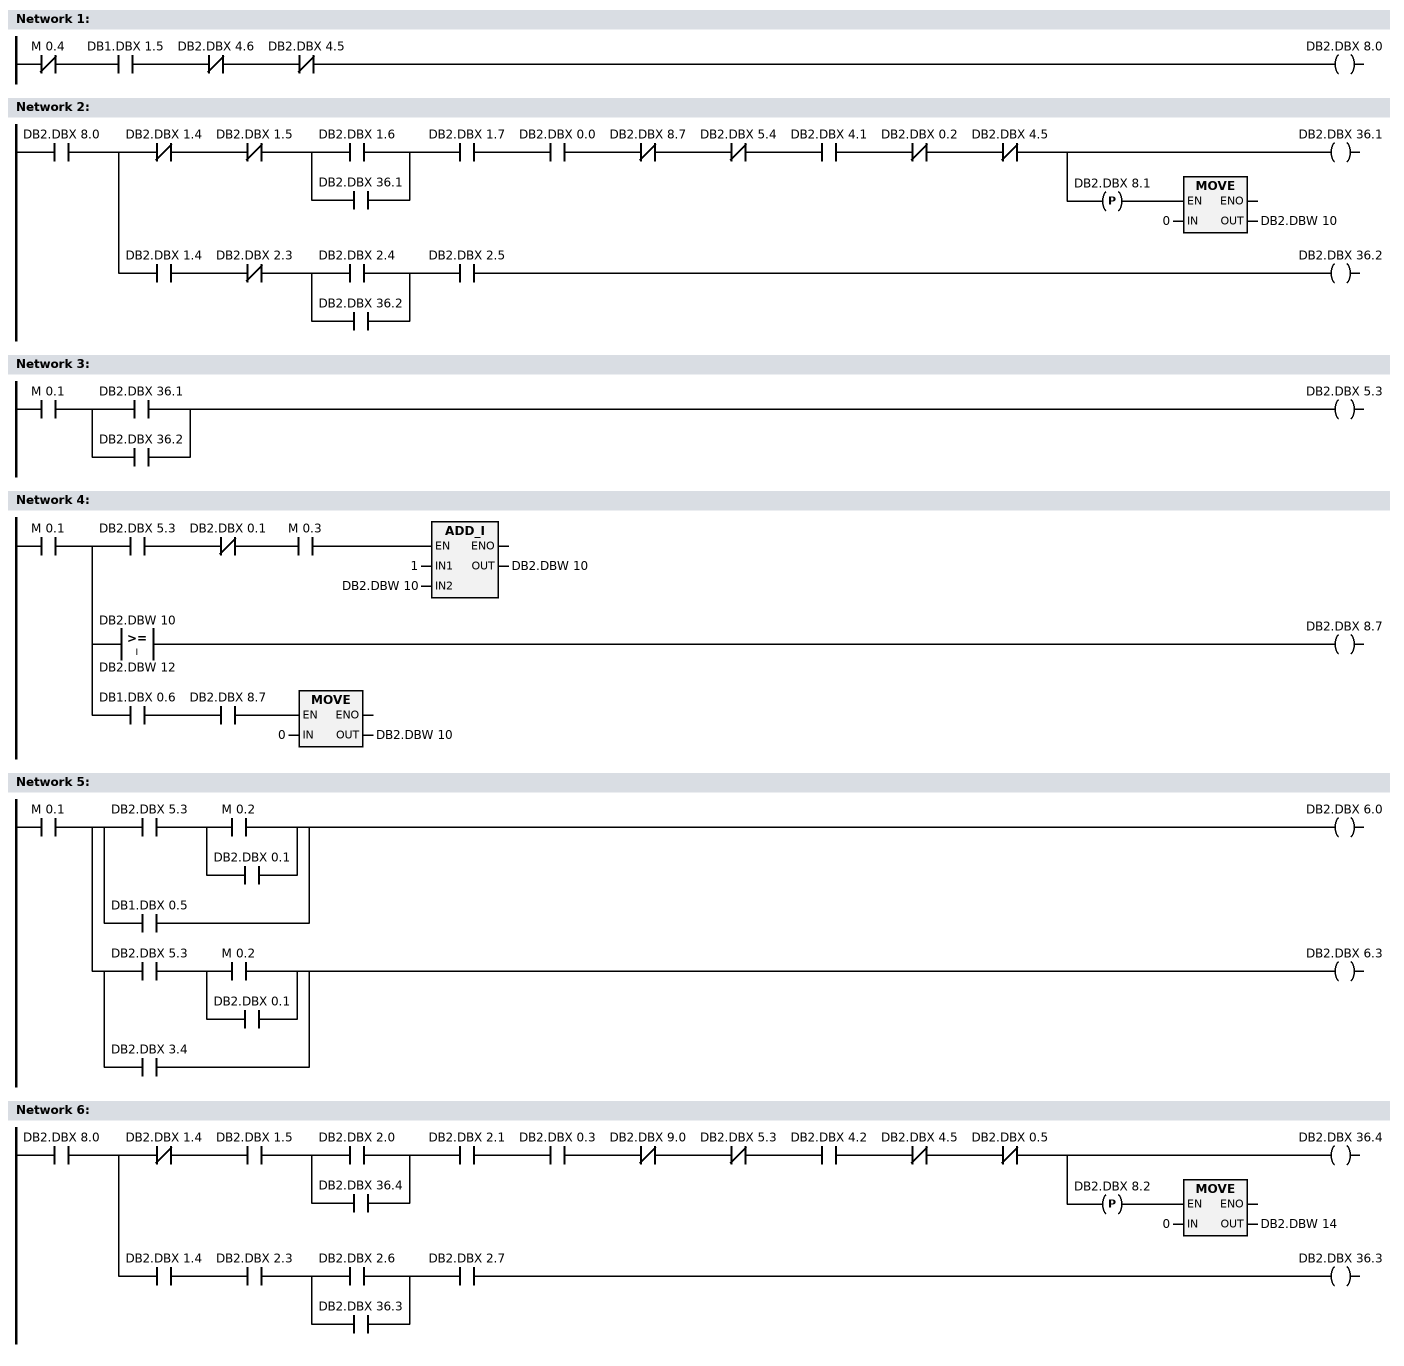
NETWORK
TITLE =
      AN    M 0.4;
      A     DB1.DBX 1.5;
      AN    DB2.DBX 4.6;
      AN    DB2.DBX 4.5;
      =     DB2.DBX 8.0;
NETWORK
TITLE =
      A     DB2.DBX 8.0;
      =     L 0.0;
      A     L 0.0;
      AN    DB2.DBX 1.4;
      AN    DB2.DBX 1.5;
      A(;
      O     DB2.DBX 1.6;
      O     DB2.DBX 36.1;
      );
      A     DB2.DBX 1.7;
      A     DB2.DBX 0.0;
      AN    DB2.DBX 8.7;
      AN    DB2.DBX 5.4;
      A     DB2.DBX 4.1;
      AN    DB2.DBX 0.2;
      AN    DB2.DBX 4.5;
      =     L 0.1;
      A     L 0.1;
      BLD   102;
      =     DB2.DBX 36.1;
      A     L 0.1;
      FP    DB2.DBX 8.1;
      JNB   M001;
      L     0;
      T     DB2.DBW 10;
M001: NOP   0;
      A     L 0.0;
      A     DB2.DBX 1.4;
      AN    DB2.DBX 2.3;
      A(;
      O     DB2.DBX 2.4;
      O     DB2.DBX 36.2;
      );
      A     DB2.DBX 2.5;
      =     DB2.DBX 36.2;
NETWORK
TITLE =
      A     M 0.1;
      A(;
      O     DB2.DBX 36.1;
      O     DB2.DBX 36.2;
      );
      =     DB2.DBX 5.3;
NETWORK
TITLE =
      A     M 0.1;
      =     L 0.0;
      A     L 0.0;
      A     DB2.DBX 5.3;
      AN    DB2.DBX 0.1;
      A     M 0.3;
      JNB   M002;
      L     1;
      L     DB2.DBW 10;
      +I;
      T     DB2.DBW 10;
M002: NOP   0;
      A     L 0.0;
      A(;
      L     DB2.DBW 10;
      L     DB2.DBW 12;
      >=I;
      );
      =     DB2.DBX 8.7;
      A     L 0.0;
      A     DB1.DBX 0.6;
      A     DB2.DBX 8.7;
      JNB   M003;
      L     0;
      T     DB2.DBW 10;
M003: NOP   0;
NETWORK
TITLE =
      A     M 0.1;
      =     L 0.0;
      A     L 0.0;
      A(;
      A     DB2.DBX 5.3;
      A(;
      O     M 0.2;
      O     DB2.DBX 0.1;
      );
      O     DB1.DBX 0.5;
      );
      =     DB2.DBX 6.0;
      A     L 0.0;
      A(;
      A     DB2.DBX 5.3;
      A(;
      O     M 0.2;
      O     DB2.DBX 0.1;
      );
      O     DB2.DBX 3.4;
      );
      =     DB2.DBX 6.3;
NETWORK
TITLE =
      A     DB2.DBX 8.0;
      =     L 0.0;
      A     L 0.0;
      AN    DB2.DBX 1.4;
      A     DB2.DBX 1.5;
      A(;
      O     DB2.DBX 2.0;
      O     DB2.DBX 36.4;
      );
      A     DB2.DBX 2.1;
      A     DB2.DBX 0.3;
      AN    DB2.DBX 9.0;
      AN    DB2.DBX 5.3;
      A     DB2.DBX 4.2;
      AN    DB2.DBX 4.5;
      AN    DB2.DBX 0.5;
      =     L 0.1;
      A     L 0.1;
      BLD   102;
      =     DB2.DBX 36.4;
      A     L 0.1;
      FP    DB2.DBX 8.2;
      JNB   M004;
      L     0;
      T     DB2.DBW 14;
M004: NOP   0;
      A     L 0.0;
      A     DB2.DBX 1.4;
      A     DB2.DBX 2.3;
      A(;
      O     DB2.DBX 2.6;
      O     DB2.DBX 36.3;
      );
      A     DB2.DBX 2.7;
      =     DB2.DBX 36.3;
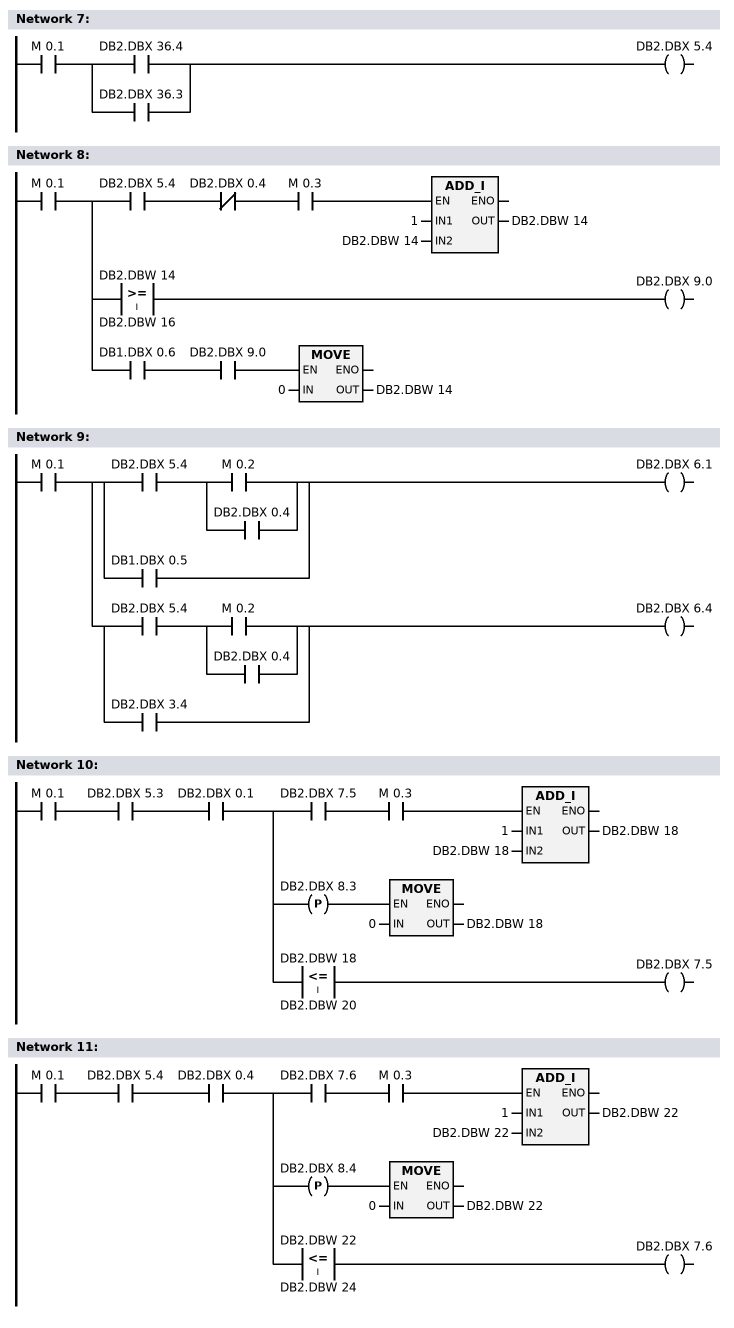
NETWORK
TITLE =
      A     M 0.1;
      A(;
      O     DB2.DBX 36.4;
      O     DB2.DBX 36.3;
      );
      =     DB2.DBX 5.4;
NETWORK
TITLE =
      A     M 0.1;
      =     L 0.0;
      A     L 0.0;
      A     DB2.DBX 5.4;
      AN    DB2.DBX 0.4;
      A     M 0.3;
      JNB   M005;
      L     1;
      L     DB2.DBW 14;
      +I;
      T     DB2.DBW 14;
M005: NOP   0;
      A     L 0.0;
      A(;
      L     DB2.DBW 14;
      L     DB2.DBW 16;
      >=I;
      );
      =     DB2.DBX 9.0;
      A     L 0.0;
      A     DB1.DBX 0.6;
      A     DB2.DBX 9.0;
      JNB   M006;
      L     0;
      T     DB2.DBW 14;
M006: NOP   0;
NETWORK
TITLE =
      A     M 0.1;
      =     L 0.0;
      A     L 0.0;
      A(;
      A     DB2.DBX 5.4;
      A(;
      O     M 0.2;
      O     DB2.DBX 0.4;
      );
      O     DB1.DBX 0.5;
      );
      =     DB2.DBX 6.1;
      A     L 0.0;
      A(;
      A     DB2.DBX 5.4;
      A(;
      O     M 0.2;
      O     DB2.DBX 0.4;
      );
      O     DB2.DBX 3.4;
      );
      =     DB2.DBX 6.4;
NETWORK
TITLE =
      A     M 0.1;
      A     DB2.DBX 5.3;
      A     DB2.DBX 0.1;
      =     L 0.0;
      A     L 0.0;
      A     DB2.DBX 7.5;
      A     M 0.3;
      JNB   M007;
      L     1;
      L     DB2.DBW 18;
      +I;
      T     DB2.DBW 18;
M007: NOP   0;
      A     L 0.0;
      FP    DB2.DBX 8.3;
      JNB   M008;
      L     0;
      T     DB2.DBW 18;
M008: NOP   0;
      A     L 0.0;
      A(;
      L     DB2.DBW 18;
      L     DB2.DBW 20;
      <=I;
      );
      =     DB2.DBX 7.5;
NETWORK
TITLE =
      A     M 0.1;
      A     DB2.DBX 5.4;
      A     DB2.DBX 0.4;
      =     L 0.0;
      A     L 0.0;
      A     DB2.DBX 7.6;
      A     M 0.3;
      JNB   M009;
      L     1;
      L     DB2.DBW 22;
      +I;
      T     DB2.DBW 22;
M009: NOP   0;
      A     L 0.0;
      FP    DB2.DBX 8.4;
      JNB   M010;
      L     0;
      T     DB2.DBW 22;
M010: NOP   0;
      A     L 0.0;
      A(;
      L     DB2.DBW 22;
      L     DB2.DBW 24;
      <=I;
      );
      =     DB2.DBX 7.6;
